C07168=1017.752,24.805,-122.391,-24.214,21.497,-42.553
C07169=1017.754,24.405,-122.357,-24.213,21.497,-42.558
C07170=1017.755,24.022,-122.323,-24.213,21.498,-42.562
C07171=1017.756,23.692,-122.294,-24.213,21.498,-42.564
C07172=1017.757,23.420,-122.270,-24.212,21.498,-42.567
C07173=1017.759,23.186,-122.250,-24.211,21.499,-42.573
C07174=1017.759,22.953,-122.230,-24.211,21.500,-42.577
C07175=1017.760,22.687,-122.207,-24.211,21.500,-42.580
C07176=1017.761,22.366,-122.179,-24.210,21.500,-42.584
C07177=1017.763,21.991,-122.147,-24.210,21.501,-42.586
C07178=1017.764,21.577,-122.111,-24.209,21.501,-42.593
C07179=1017.765,21.333,-122.089,-24.208,21.501,-42.597
C07180=1017.766,21.060,-122.066,-24.208,21.502,-42.599
C07181=1017.767,20.769,-122.041,-24.207,21.501,-42.602
C07182=1017.768,20.472,-122.015,-24.207,21.501,-42.604
C07183=1017.769,20.185,-121.990,-24.207,21.503,-42.606
C07184=1017.770,19.919,-121.966,-24.206,21.502,-42.610
C07185=1017.771,19.682,-121.946,-24.206,21.503,-42.613
C07186=1017.771,19.472,-121.927,-24.205,21.503,-42.617
C07187=1017.773,19.075,-121.894,-24.205,21.503,-42.622
C07188=1017.775,18.678,-121.859,-24.204,21.503,-42.626
C07189=1017.776,18.282,-121.824,-24.203,21.504,-42.632
C07190=1017.777,17.887,-121.790,-24.203,21.505,-42.635
C07191=1017.779,17.493,-121.757,-24.202,21.505,-42.641
C07192=1017.780,17.099,-121.723,-24.201,21.505,-42.646
C07193=1017.781,16.707,-121.689,-24.201,21.506,-42.650
C07194=1017.782,16.316,-121.655,-24.200,21.506,-42.656
C07195=1017.783,15.924,-121.622,-24.200,21.507,-42.659
C07196=1017.785,15.533,-121.587,-24.199,21.507,-42.665
C07197=1017.786,15.145,-121.554,-24.198,21.508,-42.670
C07198=1017.787,14.755,-121.520,-24.198,21.508,-42.674
C07199=1017.788,14.367,-121.487,-24.197,21.509,-42.680
C07200=1017.789,13.980,-121.454,-24.196,21.509,-42.683
C07201=1017.790,13.593,-121.420,-24.196,21.509,-42.689
C07202=1017.792,13.206,-121.387,-24.195,21.511,-42.693
C07203=1017.793,12.819,-121.354,-24.194,21.510,-42.698
C07204=1017.793,12.432,-121.321,-24.193,21.510,-42.703
C07205=1017.795,12.046,-121.287,-24.193,21.512,-42.707
C07206=1017.795,11.659,-121.254,-24.192,21.511,-42.713
C07207=1017.796,11.274,-121.221,-24.192,21.512,-42.716
C07208=1017.798,10.891,-121.188,-24.191,21.513,-42.722
C07209=1017.799,10.510,-121.156,-24.191,21.513,-42.726
C07210=1017.799,10.132,-121.123,-24.190,21.513,-42.731
C07211=1017.800,9.756,-121.091,-24.189,21.514,-42.737
C07212=1017.802,9.379,-121.059,-24.189,21.514,-42.740
C07213=1017.802,9.003,-121.027,-24.188,21.515,-42.746
C07214=1017.804,8.625,-120.994,-24.187,21.515,-42.751
C07215=1017.805,8.245,-120.962,-24.187,21.516,-42.755
C07216=1017.805,7.861,-120.929,-24.186,21.516,-42.761
C07217=1017.806,7.473,-120.896,-24.185,21.517,-42.764
C07218=1017.807,7.082,-120.862,-24.185,21.517,-42.770
C07219=1017.807,6.690,-120.829,-24.184,21.517,-42.775
C07220=1017.809,6.297,-120.796,-24.183,21.519,-42.779
C07221=1017.810,5.903,-120.762,-24.182,21.518,-42.785
C07222=1017.810,5.508,-120.728,-24.182,21.519,-42.790
C07223=1017.811,5.114,-120.695,-24.181,21.520,-42.794
C07224=1017.811,4.719,-120.661,-24.180,21.519,-42.799
C07225=1017.812,4.322,-120.628,-24.180,21.520,-42.805
C07226=1017.814,3.933,-120.595,-24.179,21.521,-42.809
C07227=1017.814,3.574,-120.564,-24.179,21.521,-42.812
C07228=1017.815,3.246,-120.536,-24.178,21.521,-42.817
C07229=1017.815,2.933,-120.509,-24.177,21.522,-42.823
C07230=1017.816,2.610,-120.482,-24.177,21.522,-42.827
C07231=1017.816,2.257,-120.453,-24.176,21.523,-42.833
C07232=1017.817,1.871,-120.419,-24.175,21.524,-42.836
C07233=1017.818,1.474,-120.386,-24.175,21.523,-42.841
C07234=1017.819,1.074,-120.352,-24.174,21.525,-42.846
C07235=1017.818,0.675,-120.318,-24.173,21.525,-42.851
C07236=1017.819,0.273,-120.284,-24.173,21.525,-42.857
C07237=1017.820,-0.130,-120.250,-24.172,21.525,-42.862
C07238=1017.821,-0.537,-120.216,-24.171,21.526,-42.867
C07239=1017.821,-0.945,-120.181,-24.171,21.527,-42.872
C07240=1017.822,-1.354,-120.147,-24.170,21.527,-42.877
C07241=1017.822,-1.767,-120.112,-24.169,21.528,-42.882
C07242=1017.823,-2.182,-120.076,-24.169,21.529,-42.888
C07243=1017.824,-2.599,-120.042,-24.168,21.529,-42.893
C07244=1017.824,-3.018,-120.007,-24.167,21.529,-42.899
C07245=1017.824,-3.439,-119.971,-24.166,21.530,-42.904
C07246=1017.824,-3.651,-119.953,-24.166,21.530,-42.908
C07247=1017.825,-3.863,-119.936,-24.165,21.530,-42.910
C07248=1017.824,-4.077,-119.918,-24.165,21.530,-42.913
C07249=1017.825,-4.292,-119.899,-24.165,21.531,-42.915
C07250=1017.826,-4.508,-119.881,-24.164,21.531,-42.919
C07251=1017.826,-4.727,-119.863,-24.164,21.531,-42.921
C07252=1017.825,-4.947,-119.844,-24.163,21.532,-42.925
C07253=1017.826,-5.169,-119.826,-24.163,21.532,-42.927
C07254=1017.826,-5.391,-119.807,-24.163,21.532,-42.930
C07255=1017.826,-5.615,-119.788,-24.162,21.532,-42.934
C07256=1017.827,-5.838,-119.769,-24.162,21.533,-42.935
C07257=1017.826,-6.064,-119.751,-24.161,21.533,-42.939
C07258=1017.827,-6.287,-119.732,-24.161,21.533,-42.941
C07259=1017.827,-6.511,-119.713,-24.161,21.533,-42.944
C07260=1017.827,-6.735,-119.695,-24.160,21.534,-42.947
C07261=1017.827,-6.957,-119.676,-24.160,21.534,-42.950
C07262=1017.827,-7.178,-119.658,-24.160,21.535,-42.952
C07263=1017.827,-7.399,-119.639,-24.159,21.534,-42.956
C07264=1017.828,-7.618,-119.621,-24.159,21.535,-42.959
C07265=1017.828,-7.836,-119.603,-24.158,21.535,-42.961
C07266=1017.828,-8.053,-119.585,-24.158,21.536,-42.965
C07267=1017.828,-8.270,-119.566,-24.158,21.536,-42.967
C07268=1017.828,-8.487,-119.548,-24.157,21.536,-42.971
C07269=1017.828,-8.703,-119.530,-24.157,21.537,-42.973
C07270=1017.828,-8.919,-119.512,-24.156,21.536,-42.976
C07271=1017.829,-9.136,-119.494,-24.156,21.537,-42.980
C07272=1017.829,-9.353,-119.476,-24.156,21.537,-42.982
C07273=1017.829,-9.569,-119.458,-24.155,21.538,-42.985
C07274=1017.829,-9.786,-119.440,-24.155,21.538,-42.987
C07275=1017.829,-10.001,-119.422,-24.154,21.538,-42.991
C07276=1017.829,-10.217,-119.404,-24.154,21.539,-42.993
C07277=1017.829,-10.432,-119.386,-24.154,21.538,-42.996
C07278=1017.829,-10.647,-119.368,-24.153,21.539,-42.998
C07279=1017.829,-10.861,-119.351,-24.153,21.539,-43.002
C07280=1017.830,-11.076,-119.333,-24.152,21.539,-43.006
C07281=1017.829,-11.290,-119.314,-24.152,21.540,-43.007
C07282=1017.830,-11.503,-119.297,-24.152,21.540,-43.011
C07283=1017.829,-11.715,-119.279,-24.151,21.540,-43.013
C07284=1017.829,-11.928,-119.262,-24.151,21.540,-43.016
C07285=1017.829,-12.140,-119.244,-24.151,21.541,-43.019
C07286=1017.829,-12.351,-119.227,-24.150,21.541,-43.022
C07287=1017.829,-12.562,-119.209,-24.150,21.542,-43.024
C07288=1017.829,-12.982,-119.174,-24.149,21.542,-43.029
C07289=1017.829,-13.400,-119.140,-24.148,21.543,-43.035
C07290=1017.829,-13.813,-119.105,-24.148,21.543,-43.041
C07291=1017.830,-14.226,-119.071,-24.147,21.544,-43.046
C07292=1017.830,-14.634,-119.037,-24.146,21.544,-43.052
C07293=1017.829,-15.039,-119.003,-24.145,21.545,-43.057
C07294=1017.829,-15.442,-118.970,-24.145,21.545,-43.063
C07295=1017.829,-15.843,-118.937,-24.144,21.546,-43.068
C07296=1017.829,-16.242,-118.904,-24.143,21.546,-43.074
C07297=1017.829,-16.642,-118.871,-24.142,21.547,-43.079
C07298=1017.829,-17.039,-118.839,-24.142,21.548,-43.085
C07299=1017.829,-17.437,-118.806,-24.141,21.547,-43.090
C07300=1017.828,-17.847,-118.772,-24.140,21.548,-43.098
C07301=1017.829,-18.096,-118.752,-24.139,21.549,-43.101
C07302=1017.828,-18.384,-118.728,-24.139,21.549,-43.105
C07303=1017.828,-18.695,-118.702,-24.139,21.550,-43.107
C07304=1017.827,-19.006,-118.677,-24.139,21.550,-43.109
C07305=1017.827,-19.294,-118.653,-24.138,21.550,-43.113
C07306=1017.827,-19.543,-118.632,-24.138,21.551,-43.116
C07307=1017.827,-19.954,-118.598,-24.136,21.551,-43.123
C07308=1017.826,-20.352,-118.566,-24.136,21.552,-43.129
C07309=1017.826,-20.749,-118.534,-24.135,21.553,-43.135
C07310=1017.826,-21.147,-118.501,-24.134,21.552,-43.140
C07311=1017.825,-21.545,-118.468,-24.134,21.553,-43.146
C07312=1017.825,-21.942,-118.435,-24.133,21.554,-43.151
C07313=1017.825,-22.340,-118.403,-24.132,21.554,-43.156
C07314=1017.824,-22.737,-118.370,-24.131,21.555,-43.162
C07315=1017.824,-23.135,-118.338,-24.131,21.555,-43.168
C07316=1017.823,-23.532,-118.305,-24.130,21.556,-43.173
C07317=1017.823,-23.929,-118.273,-24.129,21.556,-43.178
C07318=1017.823,-24.327,-118.241,-24.128,21.557,-43.184
C07319=1017.822,-24.725,-118.209,-24.128,21.558,-43.190
C07320=1017.822,-25.122,-118.176,-24.127,21.558,-43.195
C07321=1017.821,-25.520,-118.144,-24.126,21.558,-43.201
C07322=1017.821,-25.918,-118.111,-24.125,21.559,-43.206
C07323=1017.820,-26.315,-118.079,-24.125,21.560,-43.212
C07324=1017.819,-26.712,-118.047,-24.124,21.560,-43.217
C07325=1017.818,-27.109,-118.014,-24.123,21.561,-43.221
C07326=1017.818,-27.507,-117.982,-24.123,21.562,-43.227
C07327=1017.818,-27.904,-117.949,-24.122,21.562,-43.232
C07328=1017.817,-28.301,-117.917,-24.121,21.562,-43.238
C07329=1017.816,-28.700,-117.885,-24.120,21.563,-43.243
C07330=1017.815,-29.097,-117.853,-24.120,21.564,-43.249
C07331=1017.814,-29.494,-117.821,-24.119,21.565,-43.255
C07332=1017.813,-29.892,-117.789,-24.118,21.565,-43.260
C07333=1017.813,-30.289,-117.757,-24.117,21.565,-43.265
C07334=1017.812,-30.686,-117.724,-24.117,21.566,-43.271
C07335=1017.811,-31.083,-117.692,-24.116,21.567,-43.277
C07336=1017.811,-31.481,-117.661,-24.115,21.568,-43.282
C07337=1017.809,-31.879,-117.628,-24.114,21.567,-43.287
C07338=1017.809,-32.276,-117.596,-24.114,21.568,-43.293
C07339=1017.808,-32.674,-117.564,-24.113,21.569,-43.299
C07340=1017.807,-33.071,-117.532,-24.112,21.570,-43.304
C07341=1017.806,-33.469,-117.500,-24.111,21.570,-43.310
C07342=1017.806,-33.866,-117.468,-24.111,21.570,-43.315
C07343=1017.804,-34.263,-117.436,-24.110,21.571,-43.321
C07344=1017.803,-34.660,-117.404,-24.109,21.571,-43.328
C07345=1017.802,-35.058,-117.372,-24.108,21.572,-43.334
C07346=1017.801,-35.456,-117.341,-24.107,21.572,-43.339
C07347=1017.800,-35.853,-117.309,-24.107,21.573,-43.344
C07348=1017.799,-36.250,-117.277,-24.106,21.573,-43.350
C07349=1017.798,-36.647,-117.245,-24.105,21.574,-43.356
C07350=1017.797,-37.044,-117.213,-24.105,21.575,-43.361
C07351=1017.796,-37.442,-117.182,-24.104,21.575,-43.366
C07352=1017.795,-37.839,-117.150,-24.103,21.576,-43.372
C07353=1017.793,-38.237,-117.118,-24.102,21.576,-43.378
C07354=1017.792,-38.634,-117.086,-24.102,21.577,-43.383
C07355=1017.791,-39.032,-117.055,-24.101,21.578,-43.389
C07356=1017.790,-39.429,-117.022,-24.100,21.578,-43.394
C07357=1017.789,-39.826,-116.991,-24.099,21.579,-43.400
C07358=1017.787,-40.223,-116.959,-24.099,21.579,-43.405
C07359=1017.787,-40.621,-116.928,-24.098,21.580,-43.411
C07360=1017.785,-41.017,-116.896,-24.097,21.581,-43.417
C07361=1017.783,-41.415,-116.864,-24.096,21.582,-43.422
C07362=1017.783,-41.813,-116.833,-24.096,21.582,-43.427
C07363=1017.781,-42.210,-116.801,-24.095,21.582,-43.433
C07364=1017.780,-42.607,-116.770,-24.094,21.583,-43.439
C07365=1017.778,-43.004,-116.738,-24.093,21.584,-43.444
C07366=1017.777,-43.401,-116.707,-24.092,21.584,-43.451
C07367=1017.775,-43.798,-116.676,-24.092,21.585,-43.457
C07368=1017.774,-44.195,-116.644,-24.091,21.585,-43.462
C07369=1017.772,-44.593,-116.613,-24.090,21.585,-43.468
C07370=1017.771,-44.990,-116.581,-24.089,21.586,-43.473
C07371=1017.769,-45.387,-116.550,-24.089,21.587,-43.479
C07372=1017.768,-45.785,-116.519,-24.088,21.588,-43.485
C07373=1017.766,-46.182,-116.487,-24.087,21.589,-43.490
C07374=1017.765,-46.579,-116.456,-24.086,21.588,-43.496
C07375=1017.764,-46.976,-116.425,-24.086,21.589,-43.501
C07376=1017.762,-47.373,-116.393,-24.085,21.590,-43.507
C07377=1017.760,-47.770,-116.362,-24.084,21.591,-43.512
C07378=1017.758,-48.167,-116.330,-24.084,21.592,-43.518
C07379=1017.757,-48.565,-116.299,-24.083,21.592,-43.525
C07380=1017.755,-48.962,-116.268,-24.082,21.592,-43.531
C07381=1017.753,-49.358,-116.237,-24.081,21.592,-43.536
C07382=1017.752,-49.756,-116.206,-24.080,21.593,-43.542
C07383=1017.749,-50.153,-116.175,-24.080,21.594,-43.547
C07384=1017.748,-50.550,-116.143,-24.079,21.595,-43.553
C07385=1017.747,-50.947,-116.112,-24.078,21.595,-43.558
C07386=1017.744,-51.344,-116.081,-24.077,21.596,-43.564
C07387=1017.742,-51.740,-116.050,-24.077,21.597,-43.570
C07388=1017.741,-52.138,-116.019,-24.076,21.598,-43.575
C07389=1017.739,-52.534,-115.988,-24.075,21.598,-43.581
C07390=1017.737,-52.931,-115.957,-24.074,21.598,-43.588
C07391=1017.735,-53.328,-115.926,-24.073,21.599,-43.593
C07392=1017.733,-53.725,-115.896,-24.073,21.599,-43.599
C07393=1017.731,-54.122,-115.865,-24.072,21.600,-43.604
C07394=1017.729,-54.519,-115.833,-24.071,21.601,-43.610
C07395=1017.727,-54.916,-115.803,-24.071,21.602,-43.616
C07396=1017.725,-55.313,-115.772,-24.070,21.603,-43.621
C07397=1017.723,-55.711,-115.741,-24.069,21.602,-43.627
C07398=1017.721,-56.108,-115.710,-24.068,21.603,-43.632
C07399=1017.718,-56.505,-115.679,-24.067,21.603,-43.639
C07400=1017.717,-56.904,-115.648,-24.067,21.604,-43.645
C07401=1017.714,-57.302,-115.617,-24.066,21.605,-43.651
C07402=1017.713,-57.701,-115.586,-24.065,21.606,-43.656
C07403=1017.711,-58.100,-115.556,-24.064,21.606,-43.662
C07404=1017.708,-58.500,-115.525,-24.064,21.607,-43.667
C07405=1017.706,-58.900,-115.493,-24.063,21.608,-43.673
C07406=1017.703,-59.300,-115.462,-24.062,21.608,-43.680
C07407=1017.701,-59.702,-115.431,-24.061,21.609,-43.686
C07408=1017.699,-60.104,-115.401,-24.061,21.610,-43.691
C07409=1017.697,-60.506,-115.369,-24.060,21.610,-43.697
C07410=1017.694,-60.909,-115.338,-24.059,21.610,-43.702
C07411=1017.691,-61.313,-115.307,-24.058,21.611,-43.708
C07412=1017.690,-61.717,-115.276,-24.057,21.611,-43.715
C07413=1017.687,-62.121,-115.245,-24.057,21.612,-43.720
C07414=1017.684,-62.527,-115.213,-24.056,21.613,-43.726
C07415=1017.682,-62.932,-115.182,-24.055,21.614,-43.732
C07416=1017.679,-63.339,-115.151,-24.054,21.615,-43.737
C07417=1017.677,-63.745,-115.120,-24.053,21.615,-43.744
C07418=1017.674,-64.153,-115.089,-24.053,21.615,-43.750
C07419=1017.671,-64.560,-115.057,-24.052,21.616,-43.756
C07420=1017.669,-64.969,-115.026,-24.051,21.617,-43.761
C07421=1017.667,-65.377,-114.994,-24.050,21.617,-43.768
C07422=1017.664,-65.786,-114.964,-24.049,21.618,-43.774
C07423=1017.661,-66.195,-114.932,-24.049,21.619,-43.780
C07424=1017.659,-66.604,-114.901,-24.048,21.620,-43.785
C07425=1017.656,-67.014,-114.870,-24.047,21.620,-43.791
C07426=1017.653,-67.424,-114.838,-24.046,21.621,-43.798
C07427=1017.650,-67.834,-114.807,-24.046,21.621,-43.804
C07428=1017.647,-68.244,-114.776,-24.045,21.622,-43.809
C07429=1017.644,-68.655,-114.744,-24.044,21.623,-43.815
C07430=1017.641,-69.066,-114.714,-24.043,21.623,-43.822
C07431=1017.638,-69.476,-114.682,-24.042,21.624,-43.827
C07432=1017.636,-69.888,-114.650,-24.042,21.625,-43.833
C07433=1017.633,-70.298,-114.619,-24.041,21.625,-43.839
C07434=1017.630,-70.710,-114.588,-24.040,21.626,-43.846
C07435=1017.626,-71.121,-114.557,-24.039,21.626,-43.851
C07436=1017.623,-71.532,-114.525,-24.039,21.627,-43.857
C07437=1017.621,-71.942,-114.495,-24.038,21.628,-43.865
C07438=1017.617,-72.353,-114.463,-24.037,21.629,-43.870
C07439=1017.614,-72.764,-114.432,-24.036,21.630,-43.876
C07440=1017.612,-73.175,-114.401,-24.035,21.631,-43.881
C07441=1017.608,-73.586,-114.370,-24.034,21.631,-43.888
C07442=1017.605,-73.996,-114.340,-24.034,21.632,-43.894
C07443=1017.601,-74.407,-114.308,-24.033,21.632,-43.900
C07444=1017.599,-74.817,-114.277,-24.032,21.633,-43.905
C07445=1017.595,-75.226,-114.246,-24.031,21.633,-43.912
C07446=1017.591,-75.636,-114.215,-24.031,21.634,-43.918
C07447=1017.589,-76.046,-114.184,-24.030,21.635,-43.924
C07448=1017.585,-76.456,-114.153,-24.029,21.636,-43.929
C07449=1017.582,-76.865,-114.123,-24.028,21.636,-43.936
C07450=1017.579,-77.273,-114.092,-24.027,21.637,-43.942
C07451=1017.575,-77.681,-114.061,-24.027,21.637,-43.948
C07452=1017.572,-78.090,-114.030,-24.026,21.638,-43.953
C07453=1017.568,-78.497,-114.000,-24.025,21.638,-43.960
C07454=1017.564,-78.905,-113.970,-24.024,21.639,-43.966
C07455=1017.561,-79.311,-113.939,-24.023,21.640,-43.972
C07456=1017.557,-79.718,-113.908,-24.023,21.641,-43.977
C07457=1017.554,-80.124,-113.878,-24.022,21.641,-43.984
C07458=1017.551,-80.528,-113.848,-24.021,21.642,-43.990
C07459=1017.547,-80.932,-113.818,-24.020,21.643,-43.995
C07460=1017.543,-81.337,-113.787,-24.020,21.643,-44.001
C07461=1017.539,-81.739,-113.757,-24.019,21.644,-44.007
C07462=1017.536,-82.142,-113.727,-24.018,21.644,-44.014
C07463=1017.532,-82.545,-113.697,-24.017,21.645,-44.019
C07464=1017.528,-82.946,-113.667,-24.016,21.646,-44.025
C07465=1017.525,-83.347,-113.638,-24.016,21.647,-44.031
C07466=1017.521,-83.747,-113.607,-24.015,21.648,-44.036
C07467=1017.518,-84.148,-113.578,-24.014,21.648,-44.043
C07468=1017.514,-84.553,-113.548,-24.013,21.649,-44.049
C07469=1017.511,-84.777,-113.531,-24.013,21.649,-44.053
C07470=1017.509,-85.018,-113.513,-24.012,21.650,-44.056
C07471=1017.507,-85.271,-113.494,-24.012,21.649,-44.060
C07472=1017.504,-85.526,-113.475,-24.012,21.650,-44.062
C07473=1017.502,-85.772,-113.457,-24.011,21.650,-44.065
C07474=1017.499,-86.001,-113.440,-24.011,21.651,-44.069
C07475=1017.496,-86.411,-113.409,-24.010,21.652,-44.077
C07476=1017.492,-86.799,-113.381,-24.009,21.652,-44.082
C07477=1017.488,-87.179,-113.353,-24.008,21.652,-44.087
C07478=1017.485,-87.551,-113.325,-24.007,21.653,-44.093
C07479=1017.481,-87.923,-113.297,-24.007,21.654,-44.099
C07480=1017.477,-88.299,-113.270,-24.006,21.655,-44.104
C07481=1017.474,-88.706,-113.240,-24.005,21.656,-44.112
C07482=1017.470,-88.954,-113.221,-24.005,21.656,-44.116
C07483=1017.468,-89.228,-113.201,-24.004,21.657,-44.117
C07484=1017.464,-89.512,-113.180,-24.004,21.656,-44.121
C07485=1017.461,-89.787,-113.159,-24.003,21.657,-44.124
C07486=1017.459,-90.037,-113.141,-24.003,21.657,-44.128
C07487=1017.457,-90.256,-113.125,-24.002,21.658,-44.132
C07488=1017.453,-90.652,-113.096,-24.002,21.659,-44.138
C07489=1017.449,-91.045,-113.067,-24.001,21.659,-44.145
C07490=1017.444,-91.438,-113.038,-24.000,21.660,-44.150
C07491=1017.440,-91.830,-113.009,-23.999,21.660,-44.156
C07492=1017.436,-92.222,-112.980,-23.999,21.661,-44.162
C07493=1017.432,-92.612,-112.951,-23.998,21.662,-44.167
C07494=1017.428,-93.002,-112.923,-23.997,21.663,-44.173
C07495=1017.424,-93.391,-112.894,-23.996,21.664,-44.178
C07496=1017.419,-93.780,-112.866,-23.996,21.664,-44.184
C07497=1017.415,-94.168,-112.837,-23.995,21.664,-44.189
C07498=1017.411,-94.554,-112.809,-23.994,21.665,-44.195
C07499=1017.407,-94.941,-112.781,-23.994,21.666,-44.200
C07500=1017.402,-95.326,-112.752,-23.993,21.666,-44.207
C07501=1017.398,-95.711,-112.724,-23.992,21.667,-44.213
C07502=1017.393,-96.096,-112.696,-23.991,21.668,-44.219
C07503=1017.389,-96.480,-112.668,-23.990,21.668,-44.224
C07504=1017.385,-96.863,-112.640,-23.990,21.669,-44.230
C07505=1017.380,-97.247,-112.612,-23.989,21.669,-44.235
C07506=1017.376,-97.630,-112.583,-23.988,21.670,-44.241
C07507=1017.371,-98.014,-112.555,-23.988,21.671,-44.246
C07508=1017.367,-98.396,-112.528,-23.987,21.672,-44.252
C07509=1017.363,-98.780,-112.500,-23.986,21.673,-44.258
C07510=1017.358,-99.164,-112.472,-23.985,21.673,-44.263
C07511=1017.353,-99.547,-112.444,-23.985,21.673,-44.268
C07512=1017.348,-99.932,-112.416,-23.984,21.674,-44.274
C07513=1017.345,-100.316,-112.388,-23.983,21.675,-44.280
C07514=1017.339,-100.701,-112.360,-23.982,21.676,-44.285
C07515=1017.334,-101.086,-112.332,-23.982,21.677,-44.291
C07516=1017.330,-101.473,-112.304,-23.981,21.676,-44.296
C07517=1017.325,-101.861,-112.276,-23.980,21.677,-44.302
C07518=1017.320,-102.248,-112.248,-23.980,21.678,-44.307
C07519=1017.315,-102.636,-112.219,-23.979,21.678,-44.314
C07520=1017.310,-103.026,-112.192,-23.978,21.679,-44.320
C07521=1017.306,-103.416,-112.163,-23.977,21.680,-44.326
C07522=1017.301,-103.806,-112.135,-23.976,21.681,-44.331
C07523=1017.296,-104.197,-112.106,-23.976,21.682,-44.337
C07524=1017.290,-104.588,-112.078,-23.975,21.681,-44.342
C07525=1017.285,-104.981,-112.050,-23.974,21.682,-44.348
C07526=1017.280,-105.373,-112.022,-23.974,21.683,-44.353
C07527=1017.275,-105.765,-111.993,-23.973,21.684,-44.359
C07528=1017.270,-106.158,-111.965,-23.972,21.685,-44.365
C07529=1017.265,-106.552,-111.936,-23.971,21.686,-44.370
C07530=1017.260,-106.944,-111.907,-23.971,21.686,-44.376
C07531=1017.255,-107.337,-111.879,-23.970,21.687,-44.383
C07532=1017.249,-107.730,-111.851,-23.969,21.687,-44.388
C07533=1017.244,-108.123,-111.822,-23.968,21.688,-44.394
C07534=1017.238,-108.516,-111.794,-23.968,21.688,-44.399
C07535=1017.233,-108.909,-111.766,-23.967,21.689,-44.405
C07536=1017.227,-109.301,-111.738,-23.966,21.690,-44.411
C07537=1017.222,-109.695,-111.710,-23.965,21.691,-44.416
C07538=1017.217,-110.088,-111.682,-23.965,21.691,-44.422
C07539=1017.211,-110.481,-111.653,-23.964,21.692,-44.427
C07540=1017.205,-110.873,-111.625,-23.963,21.693,-44.433
C07541=1017.199,-111.266,-111.596,-23.963,21.694,-44.439
C07542=1017.194,-111.659,-111.568,-23.962,21.694,-44.446
C07543=1017.188,-112.051,-111.540,-23.961,21.694,-44.451
C07544=1017.183,-112.444,-111.512,-23.960,21.695,-44.456
C07545=1017.177,-112.836,-111.484,-23.959,21.696,-44.462
C07546=1017.172,-113.229,-111.456,-23.959,21.696,-44.468
C07547=1017.165,-113.622,-111.428,-23.958,21.697,-44.473
C07548=1017.160,-114.015,-111.400,-23.957,21.698,-44.479
C07549=1017.154,-114.407,-111.371,-23.957,21.699,-44.485
C07550=1017.148,-114.800,-111.344,-23.956,21.700,-44.490
C07551=1017.143,-115.192,-111.315,-23.955,21.701,-44.496
C07552=1017.137,-115.584,-111.287,-23.954,21.700,-44.501
C07553=1017.131,-115.977,-111.260,-23.954,21.701,-44.507
C07554=1017.125,-116.369,-111.232,-23.953,21.702,-44.512
C07555=1017.118,-116.762,-111.203,-23.952,21.703,-44.518
C07556=1017.113,-117.154,-111.176,-23.952,21.704,-44.523
C07557=1017.107,-117.546,-111.148,-23.951,21.705,-44.529
C07558=1017.100,-117.938,-111.120,-23.950,21.705,-44.536
C07559=1017.095,-118.331,-111.092,-23.949,21.705,-44.541
C07560=1017.089,-118.723,-111.064,-23.948,21.706,-44.547
C07561=1017.082,-119.115,-111.036,-23.948,21.706,-44.553
C07562=1017.077,-119.508,-111.009,-23.947,21.707,-44.558
C07563=1017.070,-119.900,-110.980,-23.946,21.708,-44.564
C07564=1017.064,-120.292,-110.952,-23.946,21.709,-44.569
C07565=1017.057,-120.684,-110.924,-23.945,21.710,-44.575
C07566=1017.051,-121.077,-110.897,-23.944,21.710,-44.580
C07567=1017.045,-121.469,-110.869,-23.943,21.710,-44.586
C07568=1017.039,-121.861,-110.841,-23.943,21.711,-44.591
C07569=1017.032,-122.253,-110.813,-23.942,21.712,-44.597
C07570=1017.026,-122.645,-110.785,-23.941,21.713,-44.603
C07571=1017.019,-123.037,-110.757,-23.941,21.714,-44.608
C07572=1017.013,-123.430,-110.730,-23.940,21.715,-44.614
C07573=1017.006,-123.821,-110.702,-23.939,21.714,-44.619
C07574=1017.000,-124.214,-110.674,-23.939,21.715,-44.625
C07575=1016.993,-124.605,-110.647,-23.938,21.716,-44.630
C07576=1016.986,-124.997,-110.619,-23.937,21.717,-44.636
C07577=1016.979,-125.390,-110.591,-23.936,21.718,-44.642
C07578=1016.973,-125.753,-110.566,-23.936,21.718,-44.647
C07579=1016.966,-126.173,-110.536,-23.935,21.719,-44.652
C07580=1016.959,-126.565,-110.508,-23.934,21.719,-44.658
C07581=1016.953,-126.957,-110.480,-23.934,21.720,-44.664
C07582=1016.946,-127.349,-110.452,-23.933,21.721,-44.669
C07583=1016.939,-127.742,-110.425,-23.932,21.722,-44.675
C07584=1016.932,-128.133,-110.398,-23.932,21.723,-44.680
C07585=1016.925,-128.525,-110.370,-23.931,21.723,-44.686
C07586=1016.918,-128.917,-110.343,-23.930,21.723,-44.691
C07587=1016.911,-129.309,-110.315,-23.929,21.724,-44.697
C07588=1016.904,-129.701,-110.287,-23.929,21.725,-44.703
C07589=1016.897,-130.093,-110.260,-23.928,21.726,-44.708
C07590=1016.890,-130.484,-110.232,-23.927,21.727,-44.714
C07591=1016.882,-130.876,-110.204,-23.926,21.727,-44.719
C07592=1016.875,-131.268,-110.177,-23.926,21.728,-44.725
C07593=1016.868,-131.659,-110.149,-23.925,21.728,-44.730
C07594=1016.861,-132.052,-110.121,-23.924,21.729,-44.736
C07595=1016.853,-132.443,-110.094,-23.924,21.730,-44.741
C07596=1016.846,-132.835,-110.067,-23.923,21.730,-44.747
C07597=1016.839,-133.227,-110.039,-23.922,21.731,-44.752
C07598=1016.831,-133.619,-110.012,-23.922,21.732,-44.758
C07599=1016.825,-134.011,-109.984,-23.921,21.732,-44.763
C07600=1017.216,-133.982,-110.228,-23.921,21.732,-44.763
C07601=1017.222,-133.590,-110.256,-23.922,21.732,-44.758
C07602=1017.230,-133.199,-110.283,-23.922,21.731,-44.752
C07603=1017.237,-132.807,-110.310,-23.923,21.730,-44.747
C07604=1017.244,-132.415,-110.338,-23.924,21.730,-44.741
C07605=1017.252,-132.023,-110.365,-23.924,21.729,-44.736
C07606=1017.259,-131.632,-110.393,-23.925,21.728,-44.730
C07607=1017.266,-131.240,-110.420,-23.926,21.728,-44.725
C07608=1017.272,-130.848,-110.448,-23.926,21.727,-44.719
C07609=1017.279,-130.456,-110.475,-23.927,21.727,-44.714
C07610=1017.286,-130.064,-110.502,-23.928,21.726,-44.708
C07611=1017.293,-129.672,-110.530,-23.929,21.725,-44.703
C07612=1017.299,-129.281,-110.557,-23.929,21.724,-44.697
C07613=1017.306,-128.889,-110.585,-23.930,21.723,-44.691
C07614=1017.314,-128.497,-110.613,-23.931,21.723,-44.686
C07615=1017.321,-128.105,-110.640,-23.932,21.723,-44.680
C07616=1017.327,-127.713,-110.667,-23.932,21.722,-44.675
C07617=1017.334,-127.321,-110.694,-23.933,21.721,-44.669
C07618=1017.341,-126.929,-110.722,-23.934,21.720,-44.664
C07619=1017.347,-126.537,-110.750,-23.934,21.719,-44.658
C07620=1017.354,-126.145,-110.778,-23.935,21.719,-44.652
C07621=1017.360,-125.753,-110.804,-23.936,21.719,-44.647
C07622=1017.366,-125.361,-110.832,-23.936,21.718,-44.642
C07623=1017.373,-124.969,-110.860,-23.937,21.717,-44.636
C07624=1017.380,-124.577,-110.888,-23.938,21.716,-44.630
C07625=1017.386,-124.185,-110.916,-23.939,21.715,-44.625
C07626=1017.393,-123.793,-110.942,-23.939,21.714,-44.619
C07627=1017.399,-123.401,-110.971,-23.940,21.715,-44.614
C07628=1017.406,-123.009,-110.998,-23.941,21.714,-44.608
C07629=1017.411,-122.617,-111.026,-23.941,21.713,-44.603
C07630=1017.418,-122.225,-111.054,-23.942,21.712,-44.597
C07631=1017.424,-121.833,-111.081,-23.943,21.711,-44.591
C07632=1017.430,-121.441,-111.109,-23.943,21.710,-44.586
C07633=1017.436,-121.048,-111.137,-23.944,21.710,-44.580
C07634=1017.442,-120.656,-111.165,-23.945,21.710,-44.575
C07635=1017.449,-120.264,-111.192,-23.946,21.709,-44.569
C07636=1017.455,-119.872,-111.220,-23.946,21.708,-44.564
C07637=1017.461,-119.480,-111.248,-23.947,21.707,-44.558
C07638=1017.467,-119.087,-111.275,-23.948,21.706,-44.553
C07639=1017.473,-118.695,-111.303,-23.948,21.706,-44.547
C07640=1017.479,-118.303,-111.332,-23.949,21.705,-44.541
C07641=1017.484,-117.911,-111.359,-23.950,21.705,-44.536
C07642=1017.490,-117.519,-111.387,-23.951,21.705,-44.529
C07643=1017.496,-117.126,-111.414,-23.952,21.704,-44.523
C07644=1017.502,-116.734,-111.442,-23.952,21.703,-44.518
C07645=1017.508,-116.342,-111.470,-23.953,21.702,-44.512
C07646=1017.513,-115.949,-111.498,-23.954,21.701,-44.507
C07647=1017.519,-115.557,-111.526,-23.954,21.700,-44.501
C07648=1017.525,-115.165,-111.554,-23.955,21.701,-44.496
C07649=1017.530,-114.772,-111.582,-23.956,21.700,-44.490
C07650=1017.536,-114.380,-111.610,-23.957,21.699,-44.485
C07651=1017.542,-113.987,-111.637,-23.957,21.698,-44.479
C07652=1017.548,-113.595,-111.666,-23.958,21.697,-44.473
C07653=1017.553,-113.202,-111.694,-23.959,21.696,-44.468
C07654=1017.559,-112.810,-111.722,-23.959,21.696,-44.462
C07655=1017.565,-112.416,-111.750,-23.960,21.695,-44.456
C07656=1017.571,-112.024,-111.779,-23.961,21.694,-44.451
C07657=1017.576,-111.631,-111.807,-23.962,21.694,-44.446
C07658=1017.581,-111.238,-111.834,-23.963,21.694,-44.439
C07659=1017.587,-110.846,-111.863,-23.963,21.693,-44.433
C07660=1017.592,-110.453,-111.891,-23.964,21.692,-44.427
C07661=1017.598,-110.060,-111.918,-23.965,21.691,-44.422
C07662=1017.603,-109.668,-111.947,-23.965,21.691,-44.416
C07663=1017.608,-109.275,-111.975,-23.966,21.690,-44.411
C07664=1017.613,-108.882,-112.003,-23.967,21.689,-44.405
C07665=1017.618,-108.489,-112.031,-23.968,21.688,-44.399
C07666=1017.624,-108.096,-112.060,-23.968,21.688,-44.394
C07667=1017.629,-107.703,-112.088,-23.969,21.687,-44.388
C07668=1017.634,-107.310,-112.116,-23.970,21.687,-44.383
C07669=1017.639,-106.917,-112.144,-23.971,21.686,-44.376
C07670=1017.644,-106.524,-112.172,-23.971,21.686,-44.370
C07671=1017.650,-106.132,-112.201,-23.972,21.685,-44.365
C07672=1017.654,-105.738,-112.229,-23.973,21.684,-44.359
C07673=1017.659,-105.345,-112.257,-23.974,21.683,-44.353
C07674=1017.664,-104.953,-112.286,-23.974,21.682,-44.348
C07675=1017.669,-104.561,-112.314,-23.975,21.681,-44.342
C07676=1017.675,-104.170,-112.342,-23.976,21.682,-44.337
C07677=1017.679,-103.778,-112.371,-23.976,21.681,-44.331
C07678=1017.684,-103.388,-112.399,-23.977,21.680,-44.326
C07679=1017.689,-102.999,-112.427,-23.978,21.679,-44.320
C07680=1017.694,-102.609,-112.455,-23.979,21.678,-44.314
C07681=1017.698,-102.221,-112.483,-23.980,21.678,-44.307
C07682=1017.702,-101.833,-112.511,-23.980,21.677,-44.302
C07683=1017.708,-101.446,-112.539,-23.981,21.676,-44.296
C07684=1017.713,-101.060,-112.567,-23.982,21.677,-44.291
C07685=1017.717,-100.673,-112.595,-23.982,21.676,-44.285
C07686=1017.722,-100.288,-112.623,-23.983,21.675,-44.280
C07687=1017.726,-99.904,-112.651,-23.984,21.674,-44.274
C07688=1017.731,-99.520,-112.679,-23.985,21.673,-44.268
C07689=1017.735,-99.136,-112.707,-23.985,21.673,-44.263
C07690=1017.740,-98.753,-112.735,-23.986,21.673,-44.258
C07691=1017.744,-98.370,-112.763,-23.987,21.672,-44.252
C07692=1017.748,-97.986,-112.791,-23.988,21.671,-44.246
C07693=1017.753,-97.603,-112.819,-23.988,21.670,-44.241
C07694=1017.757,-97.220,-112.847,-23.989,21.669,-44.235
C07695=1017.762,-96.836,-112.875,-23.990,21.669,-44.230
C07696=1017.765,-96.452,-112.903,-23.990,21.668,-44.224
C07697=1017.770,-96.069,-112.930,-23.991,21.668,-44.219
C07698=1017.775,-95.684,-112.959,-23.992,21.667,-44.213
C07699=1017.779,-95.299,-112.987,-23.993,21.666,-44.207
C07700=1017.783,-94.913,-113.015,-23.994,21.666,-44.200
C07701=1017.787,-94.527,-113.043,-23.994,21.665,-44.195
C07702=1017.791,-94.140,-113.072,-23.995,21.664,-44.189
C07703=1017.795,-93.753,-113.101,-23.996,21.664,-44.184
C07704=1017.800,-93.365,-113.129,-23.996,21.664,-44.178
C07705=1017.804,-92.975,-113.157,-23.997,21.663,-44.173
C07706=1017.808,-92.585,-113.186,-23.998,21.662,-44.167
C07707=1017.813,-92.194,-113.214,-23.999,21.661,-44.162
C07708=1017.816,-91.803,-113.243,-23.999,21.660,-44.156
C07709=1017.820,-91.411,-113.272,-24.000,21.660,-44.150
C07710=1017.824,-91.018,-113.301,-24.001,21.659,-44.145
C07711=1017.828,-90.624,-113.330,-24.002,21.659,-44.138
C07712=1017.832,-90.229,-113.359,-24.002,21.658,-44.132
C07713=1017.835,-90.010,-113.375,-24.003,21.657,-44.128
C07714=1017.837,-89.760,-113.393,-24.003,21.657,-44.124
C07715=1017.840,-89.485,-113.414,-24.004,21.656,-44.121
C07716=1017.843,-89.200,-113.435,-24.004,21.657,-44.117
C07717=1017.845,-88.926,-113.455,-24.005,21.656,-44.116
C07718=1017.848,-88.679,-113.473,-24.005,21.656,-44.112
C07719=1017.852,-88.271,-113.503,-24.006,21.655,-44.104
C07720=1017.855,-87.896,-113.531,-24.007,21.654,-44.099
C07721=1017.859,-87.524,-113.559,-24.007,21.653,-44.093
C07722=1017.863,-87.151,-113.586,-24.008,21.652,-44.087
C07723=1017.866,-86.772,-113.614,-24.009,21.652,-44.082
C07724=1017.870,-86.384,-113.643,-24.010,21.652,-44.077
C07725=1017.874,-85.975,-113.673,-24.011,21.651,-44.069
C07726=1017.876,-85.745,-113.690,-24.011,21.650,-44.065
C07727=1017.878,-85.499,-113.708,-24.012,21.650,-44.062
C07728=1017.881,-85.244,-113.727,-24.012,21.649,-44.060
C07729=1017.883,-84.991,-113.746,-24.012,21.650,-44.056
C07730=1017.885,-84.750,-113.764,-24.013,21.649,-44.053
C07731=1017.887,-84.527,-113.781,-24.013,21.649,-44.049
C07732=1017.891,-84.120,-113.811,-24.014,21.648,-44.043
C07733=1017.895,-83.721,-113.840,-24.015,21.648,-44.036
C07734=1017.898,-83.320,-113.870,-24.016,21.647,-44.031
C07735=1017.902,-82.919,-113.900,-24.016,21.646,-44.025
C07736=1017.906,-82.518,-113.930,-24.017,21.645,-44.019
C07737=1017.910,-82.116,-113.960,-24.018,21.644,-44.014
C07738=1017.913,-81.713,-113.990,-24.019,21.644,-44.007
C07739=1017.917,-81.310,-114.020,-24.020,21.643,-44.001
C07740=1017.920,-80.905,-114.050,-24.020,21.643,-43.995
C07741=1017.924,-80.501,-114.080,-24.021,21.642,-43.990
C07742=1017.927,-80.096,-114.111,-24.022,21.641,-43.984
C07743=1017.930,-79.691,-114.141,-24.023,21.641,-43.977
C07744=1017.934,-79.284,-114.172,-24.023,21.640,-43.972
C07745=1017.937,-78.878,-114.202,-24.024,21.639,-43.966
C07746=1017.941,-78.470,-114.232,-24.025,21.638,-43.960
C07747=1017.945,-78.062,-114.263,-24.026,21.638,-43.953
C07748=1017.947,-77.655,-114.293,-24.027,21.637,-43.948
C07749=1017.951,-77.246,-114.324,-24.027,21.637,-43.942
C07750=1017.954,-76.837,-114.355,-24.028,21.636,-43.936
C07751=1017.957,-76.428,-114.386,-24.029,21.636,-43.929
C07752=1017.960,-76.019,-114.417,-24.030,21.635,-43.924
C07753=1017.964,-75.610,-114.447,-24.031,21.634,-43.918
C07754=1017.968,-75.200,-114.478,-24.031,21.633,-43.912
C07755=1017.970,-74.790,-114.509,-24.032,21.633,-43.905
C07756=1017.973,-74.379,-114.540,-24.033,21.632,-43.900
C07757=1017.977,-73.969,-114.571,-24.034,21.632,-43.894
C07758=1017.980,-73.559,-114.602,-24.034,21.631,-43.888
C07759=1017.983,-73.148,-114.633,-24.035,21.631,-43.881
C07760=1017.985,-72.737,-114.664,-24.036,21.630,-43.876
C07761=1017.989,-72.326,-114.696,-24.037,21.629,-43.870
C07762=1017.992,-71.915,-114.727,-24.038,21.628,-43.865
C07763=1017.995,-71.504,-114.757,-24.039,21.627,-43.857
C07764=1017.998,-71.094,-114.789,-24.039,21.626,-43.851
C07765=1018.001,-70.682,-114.820,-24.040,21.626,-43.846
C07766=1018.004,-70.272,-114.850,-24.041,21.625,-43.839
C07767=1018.007,-69.861,-114.882,-24.042,21.625,-43.833
C07768=1018.010,-69.450,-114.913,-24.042,21.624,-43.827
C07769=1018.013,-69.039,-114.944,-24.043,21.623,-43.822
C07770=1018.015,-68.628,-114.976,-24.044,21.623,-43.815
C07771=1018.018,-68.218,-115.007,-24.045,21.622,-43.809
C07772=1018.021,-67.808,-115.039,-24.046,21.621,-43.804
C07773=1018.023,-67.397,-115.069,-24.046,21.621,-43.798
C07774=1018.026,-66.987,-115.101,-24.047,21.620,-43.791
C07775=1018.029,-66.578,-115.133,-24.048,21.620,-43.785
C07776=1018.032,-66.168,-115.164,-24.049,21.619,-43.780
C07777=1018.034,-65.758,-115.195,-24.049,21.618,-43.774
C07778=1018.038,-65.350,-115.226,-24.050,21.617,-43.768
C07779=1018.040,-64.942,-115.257,-24.051,21.617,-43.761
C07780=1018.042,-64.533,-115.289,-24.052,21.616,-43.756
C07781=1018.045,-64.126,-115.320,-24.053,21.615,-43.750
C07782=1018.048,-63.719,-115.351,-24.053,21.615,-43.744
C07783=1018.050,-63.313,-115.382,-24.054,21.615,-43.737
C07784=1018.053,-62.906,-115.413,-24.055,21.614,-43.732
C07785=1018.055,-62.500,-115.444,-24.056,21.613,-43.726
C07786=1018.057,-62.095,-115.476,-24.057,21.612,-43.720
C07787=1018.060,-61.690,-115.506,-24.057,21.611,-43.715
C07788=1018.062,-61.285,-115.538,-24.058,21.611,-43.708
C07789=1018.065,-60.882,-115.569,-24.059,21.610,-43.702
C07790=1018.066,-60.479,-115.600,-24.060,21.610,-43.697
C07791=1018.069,-60.077,-115.631,-24.061,21.610,-43.691
C07792=1018.071,-59.675,-115.661,-24.061,21.609,-43.686
C07793=1018.073,-59.274,-115.693,-24.062,21.608,-43.680
C07794=1018.076,-58.874,-115.724,-24.063,21.608,-43.673
C07795=1018.078,-58.473,-115.755,-24.064,21.607,-43.667
C07796=1018.080,-58.074,-115.786,-24.064,21.606,-43.662
C07797=1018.083,-57.674,-115.817,-24.065,21.606,-43.656
C07798=1018.084,-57.275,-115.847,-24.066,21.605,-43.651
C07799=1018.087,-56.877,-115.878,-24.067,21.604,-43.645
C07800=1018.088,-56.479,-115.909,-24.067,21.603,-43.639
C07801=1018.091,-56.081,-115.940,-24.068,21.603,-43.632
C07802=1018.092,-55.683,-115.971,-24.069,21.602,-43.627
C07803=1018.095,-55.286,-116.002,-24.070,21.603,-43.621
C07804=1018.097,-54.889,-116.032,-24.071,21.602,-43.616
C07805=1018.098,-54.492,-116.064,-24.071,21.601,-43.610
C07806=1018.101,-54.095,-116.095,-24.072,21.600,-43.604
C07807=1018.103,-53.698,-116.125,-24.073,21.599,-43.599
C07808=1018.104,-53.301,-116.157,-24.073,21.599,-43.593
C07809=1018.106,-52.905,-116.188,-24.074,21.598,-43.588
C07810=1018.108,-52.507,-116.218,-24.075,21.598,-43.581
C07811=1018.110,-52.110,-116.250,-24.076,21.598,-43.575
C07812=1018.112,-51.714,-116.281,-24.077,21.597,-43.570
C07813=1018.114,-51.317,-116.311,-24.077,21.596,-43.564
C07814=1018.116,-50.920,-116.343,-24.078,21.595,-43.558
C07815=1018.117,-50.523,-116.374,-24.079,21.595,-43.553
C07816=1018.119,-50.126,-116.405,-24.080,21.594,-43.547
C07817=1018.121,-49.729,-116.436,-24.080,21.593,-43.542
C07818=1018.123,-49.332,-116.467,-24.081,21.592,-43.536
C07819=1018.124,-48.934,-116.498,-24.082,21.592,-43.531
C07820=1018.125,-48.537,-116.530,-24.083,21.592,-43.525
C07821=1018.128,-48.141,-116.561,-24.084,21.592,-43.518
C07822=1018.129,-47.743,-116.591,-24.084,21.591,-43.512
C07823=1018.130,-47.346,-116.623,-24.085,21.590,-43.507
C07824=1018.132,-46.949,-116.655,-24.086,21.589,-43.501
C07825=1018.133,-46.552,-116.685,-24.086,21.588,-43.496
C07826=1018.135,-46.155,-116.717,-24.087,21.589,-43.490
C07827=1018.137,-45.758,-116.748,-24.088,21.588,-43.485
C07828=1018.138,-45.361,-116.779,-24.089,21.587,-43.479
C07829=1018.140,-44.964,-116.811,-24.089,21.586,-43.473
C07830=1018.142,-44.566,-116.842,-24.090,21.585,-43.468
C07831=1018.143,-44.169,-116.873,-24.091,21.585,-43.462
C07832=1018.144,-43.772,-116.905,-24.092,21.585,-43.457
C07833=1018.145,-43.375,-116.937,-24.092,21.584,-43.451
C07834=1018.146,-42.977,-116.968,-24.093,21.584,-43.444
C07835=1018.148,-42.580,-117.000,-24.094,21.583,-43.439
C07836=1018.149,-42.183,-117.031,-24.095,21.582,-43.433
C07837=1018.151,-41.786,-117.062,-24.096,21.582,-43.427
C07838=1018.152,-41.389,-117.094,-24.096,21.582,-43.422
C07839=1018.153,-40.991,-117.126,-24.097,21.581,-43.417
C07840=1018.154,-40.595,-117.157,-24.098,21.580,-43.411
C07841=1018.156,-40.196,-117.189,-24.099,21.579,-43.405
C07842=1018.157,-39.799,-117.221,-24.099,21.579,-43.400
C07843=1018.159,-39.402,-117.252,-24.100,21.578,-43.394
C07844=1018.160,-39.005,-117.283,-24.101,21.578,-43.389
C07845=1018.160,-38.607,-117.315,-24.102,21.577,-43.383
C07846=1018.162,-38.210,-117.347,-24.102,21.576,-43.378
C07847=1018.163,-37.813,-117.379,-24.103,21.576,-43.372
C07848=1018.164,-37.416,-117.410,-24.104,21.575,-43.366
C07849=1018.165,-37.018,-117.442,-24.105,21.575,-43.361
C07850=1018.166,-36.620,-117.475,-24.105,21.574,-43.356
C07851=1018.168,-36.223,-117.506,-24.106,21.573,-43.350
C07852=1018.168,-35.826,-117.538,-24.107,21.573,-43.344
C07853=1018.170,-35.429,-117.570,-24.107,21.572,-43.339
C07854=1018.170,-35.031,-117.602,-24.108,21.572,-43.334
C07855=1018.171,-34.634,-117.634,-24.109,21.571,-43.328
C07856=1018.172,-34.236,-117.665,-24.110,21.571,-43.321
C07857=1018.173,-33.839,-117.697,-24.111,21.570,-43.315
C07858=1018.174,-33.442,-117.729,-24.111,21.570,-43.310
C07859=1018.175,-33.044,-117.762,-24.112,21.570,-43.304
C07860=1018.176,-32.647,-117.794,-24.113,21.569,-43.299
C07861=1018.176,-32.249,-117.825,-24.114,21.568,-43.293
C07862=1018.177,-31.852,-117.858,-24.114,21.567,-43.287
C07863=1018.178,-31.455,-117.890,-24.115,21.568,-43.282
C07864=1018.179,-31.057,-117.922,-24.116,21.567,-43.277
C07865=1018.180,-30.660,-117.954,-24.117,21.566,-43.271
C07866=1018.180,-30.263,-117.986,-24.117,21.565,-43.265
C07867=1018.181,-29.865,-118.018,-24.118,21.565,-43.260
C07868=1018.182,-29.467,-118.050,-24.119,21.565,-43.255
C07869=1018.183,-29.070,-118.082,-24.120,21.564,-43.249
C07870=1018.184,-28.673,-118.115,-24.120,21.563,-43.243
C07871=1018.184,-28.275,-118.147,-24.121,21.562,-43.238
C07872=1018.185,-27.878,-118.179,-24.122,21.562,-43.232
C07873=1018.186,-27.481,-118.211,-24.123,21.562,-43.227
C07874=1018.186,-27.083,-118.243,-24.123,21.561,-43.221
C07875=1018.187,-26.685,-118.275,-24.124,21.560,-43.217
C07876=1018.187,-26.288,-118.308,-24.125,21.560,-43.212
C07877=1018.187,-25.891,-118.340,-24.125,21.559,-43.206
C07878=1018.189,-25.493,-118.373,-24.126,21.558,-43.201
C07879=1018.189,-25.095,-118.405,-24.127,21.558,-43.195
C07880=1018.189,-24.698,-118.438,-24.128,21.558,-43.190
C07881=1018.190,-24.301,-118.470,-24.128,21.557,-43.184
C07882=1018.191,-23.903,-118.502,-24.129,21.556,-43.178
C07883=1018.191,-23.506,-118.535,-24.130,21.556,-43.173
C07884=1018.192,-23.109,-118.567,-24.131,21.555,-43.168
C07885=1018.192,-22.711,-118.600,-24.131,21.555,-43.162
C07886=1018.192,-22.313,-118.632,-24.132,21.554,-43.156
C07887=1018.192,-21.916,-118.664,-24.133,21.554,-43.151
C07888=1018.192,-21.518,-118.697,-24.134,21.553,-43.146
C07889=1018.194,-21.120,-118.730,-24.134,21.552,-43.140
C07890=1018.194,-20.723,-118.762,-24.135,21.553,-43.135
C07891=1018.194,-20.325,-118.795,-24.136,21.552,-43.129
C07892=1018.195,-19.928,-118.827,-24.136,21.551,-43.123
C07893=1018.195,-19.517,-118.862,-24.138,21.551,-43.116
C07894=1018.195,-19.268,-118.882,-24.138,21.550,-43.113
C07895=1018.195,-18.979,-118.906,-24.139,21.550,-43.109
C07896=1018.195,-18.668,-118.931,-24.139,21.550,-43.107
C07897=1018.195,-18.357,-118.957,-24.139,21.549,-43.105
C07898=1018.195,-18.070,-118.980,-24.139,21.549,-43.101
C07899=1018.196,-17.821,-119.002,-24.140,21.548,-43.098
C07900=1018.196,-17.410,-119.035,-24.141,21.547,-43.090
C07901=1018.196,-17.012,-119.067,-24.142,21.548,-43.085
C07902=1018.196,-16.615,-119.100,-24.142,21.547,-43.079
C07903=1018.196,-16.216,-119.133,-24.143,21.546,-43.074
C07904=1018.197,-15.816,-119.166,-24.144,21.546,-43.068
C07905=1018.196,-15.415,-119.199,-24.145,21.545,-43.063
C07906=1018.196,-15.012,-119.233,-24.145,21.545,-43.057
C07907=1018.196,-14.607,-119.266,-24.146,21.544,-43.052
C07908=1018.196,-14.199,-119.300,-24.147,21.544,-43.046
C07909=1018.197,-13.787,-119.334,-24.148,21.543,-43.041
C07910=1018.197,-13.373,-119.369,-24.148,21.543,-43.035
C07911=1018.197,-12.955,-119.403,-24.149,21.542,-43.029
C07912=1018.197,-12.535,-119.438,-24.150,21.542,-43.024
C07913=1018.196,-12.324,-119.455,-24.150,21.541,-43.022
C07914=1018.197,-12.113,-119.473,-24.151,21.541,-43.019
C07915=1018.197,-11.902,-119.491,-24.151,21.540,-43.016
C07916=1018.197,-11.689,-119.508,-24.151,21.540,-43.013
C07917=1018.196,-11.476,-119.526,-24.152,21.540,-43.011
C07918=1018.196,-11.263,-119.544,-24.152,21.540,-43.007
C07919=1018.197,-11.049,-119.562,-24.152,21.539,-43.006
C07920=1018.197,-10.835,-119.580,-24.153,21.539,-43.002
C07921=1018.197,-10.620,-119.597,-24.153,21.539,-42.998
C07922=1018.196,-10.406,-119.615,-24.154,21.538,-42.996
C07923=1018.196,-10.190,-119.633,-24.154,21.539,-42.993
C07924=1018.196,-9.975,-119.650,-24.154,21.538,-42.991
C07925=1018.196,-9.759,-119.669,-24.155,21.538,-42.987
C07926=1018.196,-9.543,-119.687,-24.155,21.538,-42.985
C07927=1018.196,-9.327,-119.705,-24.156,21.537,-42.982
C07928=1018.196,-9.109,-119.723,-24.156,21.537,-42.980
C07929=1018.195,-8.893,-119.741,-24.156,21.536,-42.976
C07930=1018.195,-8.677,-119.759,-24.157,21.537,-42.973
C07931=1018.196,-8.460,-119.777,-24.157,21.536,-42.971
C07932=1018.195,-8.243,-119.796,-24.158,21.536,-42.967
C07933=1018.195,-8.026,-119.814,-24.158,21.536,-42.965
C07934=1018.196,-7.810,-119.832,-24.158,21.535,-42.961
C07935=1018.195,-7.591,-119.850,-24.159,21.535,-42.959
C07936=1018.195,-7.372,-119.868,-24.159,21.534,-42.956
C07937=1018.195,-7.151,-119.887,-24.160,21.535,-42.952
C07938=1018.194,-6.930,-119.905,-24.160,21.534,-42.950
C07939=1018.195,-6.708,-119.923,-24.160,21.534,-42.947
C07940=1018.194,-6.484,-119.942,-24.161,21.533,-42.944
C07941=1018.194,-6.261,-119.961,-24.161,21.533,-42.941
C07942=1018.194,-6.037,-119.980,-24.161,21.533,-42.939
C07943=1018.194,-5.812,-119.998,-24.162,21.533,-42.935
C07944=1018.194,-5.588,-120.017,-24.162,21.532,-42.934
C07945=1018.193,-5.364,-120.036,-24.163,21.532,-42.930
C07946=1018.193,-5.142,-120.055,-24.163,21.532,-42.927
C07947=1018.193,-4.921,-120.073,-24.163,21.532,-42.925
C07948=1018.192,-4.701,-120.092,-24.164,21.531,-42.921
C07949=1018.192,-4.482,-120.110,-24.164,21.531,-42.919
C07950=1018.192,-4.265,-120.128,-24.165,21.531,-42.915
C07951=1018.192,-4.050,-120.147,-24.165,21.530,-42.913
C07952=1018.192,-3.837,-120.164,-24.165,21.530,-42.910
C07953=1018.191,-3.624,-120.182,-24.166,21.530,-42.908
C07954=1018.192,-3.413,-120.200,-24.166,21.530,-42.904
C07955=1018.190,-2.992,-120.235,-24.167,21.529,-42.899
C07956=1018.190,-2.572,-120.271,-24.168,21.529,-42.893
C07957=1018.189,-2.155,-120.306,-24.169,21.529,-42.888
C07958=1018.189,-1.740,-120.341,-24.169,21.528,-42.882
C07959=1018.189,-1.328,-120.376,-24.170,21.527,-42.877
C07960=1018.188,-0.918,-120.411,-24.171,21.527,-42.872
C07961=1018.188,-0.510,-120.445,-24.171,21.526,-42.867
C07962=1018.187,-0.104,-120.479,-24.172,21.525,-42.862
C07963=1018.187,0.300,-120.513,-24.173,21.525,-42.857
C07964=1018.186,0.701,-120.547,-24.173,21.525,-42.851
C07965=1018.185,1.101,-120.582,-24.174,21.525,-42.846
C07966=1018.185,1.500,-120.615,-24.175,21.523,-42.841
C07967=1018.184,1.898,-120.648,-24.175,21.524,-42.836
C07968=1018.184,2.283,-120.681,-24.176,21.523,-42.833
C07969=1018.183,2.637,-120.711,-24.177,21.522,-42.827
C07970=1018.182,2.959,-120.738,-24.177,21.522,-42.823
C07971=1018.182,3.273,-120.765,-24.178,21.521,-42.817
C07972=1018.181,3.601,-120.793,-24.179,21.521,-42.812
C07973=1018.180,3.959,-120.823,-24.179,21.521,-42.809
C07974=1018.180,4.349,-120.856,-24.180,21.520,-42.805
C07975=1018.179,4.745,-120.890,-24.180,21.519,-42.799
C07976=1018.178,5.140,-120.924,-24.181,21.520,-42.794
C07977=1018.178,5.535,-120.957,-24.182,21.519,-42.790
C07978=1018.177,5.930,-120.991,-24.182,21.518,-42.785
C07979=1018.176,6.323,-121.024,-24.183,21.519,-42.779
C07980=1018.175,6.716,-121.058,-24.184,21.517,-42.775
C07981=1018.174,7.109,-121.091,-24.185,21.517,-42.770
C07982=1018.173,7.499,-121.125,-24.185,21.517,-42.764
C07983=1018.173,7.888,-121.158,-24.186,21.516,-42.761
C07984=1018.171,8.271,-121.190,-24.187,21.516,-42.755
C07985=1018.170,8.652,-121.223,-24.187,21.515,-42.751
C07986=1018.170,9.030,-121.255,-24.188,21.515,-42.746
C07987=1018.169,9.406,-121.288,-24.189,21.514,-42.740
C07988=1018.168,9.782,-121.320,-24.189,21.514,-42.737
C07989=1018.167,10.159,-121.352,-24.190,21.513,-42.731
C07990=1018.166,10.537,-121.385,-24.191,21.513,-42.726
C07991=1018.165,10.917,-121.417,-24.191,21.513,-42.722
C07992=1018.164,11.300,-121.450,-24.192,21.512,-42.716
C07993=1018.163,11.686,-121.483,-24.192,21.511,-42.713
C07994=1018.162,12.073,-121.516,-24.193,21.512,-42.707
C07995=1018.161,12.459,-121.549,-24.193,21.510,-42.703
C07996=1018.160,12.845,-121.582,-24.194,21.510,-42.698
C07997=1018.159,13.232,-121.616,-24.195,21.511,-42.693
C07998=1018.158,13.620,-121.649,-24.196,21.509,-42.689
C07999=1018.157,14.006,-121.683,-24.196,21.509,-42.683
C08000=1018.155,14.394,-121.716,-24.197,21.509,-42.680
C08001=1018.154,14.782,-121.749,-24.198,21.508,-42.674
C08002=1018.153,15.171,-121.783,-24.198,21.508,-42.670
C08003=1018.151,15.560,-121.816,-24.199,21.507,-42.665
C08004=1018.151,15.951,-121.850,-24.200,21.507,-42.659
C08005=1018.150,16.342,-121.884,-24.200,21.506,-42.656
C08006=1018.148,16.734,-121.917,-24.201,21.506,-42.650
C08007=1018.147,17.126,-121.952,-24.201,21.505,-42.646
C08008=1018.146,17.519,-121.985,-24.202,21.505,-42.641
C08009=1018.144,17.914,-122.019,-24.203,21.505,-42.635
C08010=1018.143,18.308,-122.054,-24.203,21.504,-42.632
C08011=1018.142,18.705,-122.088,-24.204,21.503,-42.626
C08012=1018.141,19.101,-122.123,-24.205,21.503,-42.622
C08013=1018.139,19.498,-122.157,-24.205,21.503,-42.617
C08014=1018.139,19.710,-122.175,-24.206,21.503,-42.613
C08015=1018.138,19.946,-122.195,-24.206,21.502,-42.610
C08016=1018.137,20.211,-122.219,-24.207,21.503,-42.606
C08017=1018.136,20.499,-122.244,-24.207,21.501,-42.604
C08018=1018.134,20.795,-122.270,-24.207,21.501,-42.602
C08019=1018.133,21.087,-122.295,-24.208,21.502,-42.599
C08020=1018.133,21.359,-122.318,-24.208,21.501,-42.597
C08021=1018.131,21.604,-122.339,-24.209,21.501,-42.593
C08022=1018.130,22.017,-122.376,-24.210,21.501,-42.586
C08023=1018.129,22.392,-122.409,-24.210,21.500,-42.584
C08024=1018.128,22.715,-122.436,-24.211,21.500,-42.580
C08025=1018.127,22.980,-122.459,-24.211,21.500,-42.577
C08026=1018.126,23.212,-122.479,-24.211,21.499,-42.573
C08027=1018.125,23.447,-122.500,-24.212,21.498,-42.567
C08028=1018.124,23.718,-122.524,-24.213,21.498,-42.564
C08029=1018.123,24.049,-122.552,-24.213,21.498,-42.562
C08030=1018.121,24.432,-122.585,-24.213,21.497,-42.558
C08031=1018.119,24.831,-122.620,-24.214,21.497,-42.553
C08032=1018.118,25.230,-122.655,-24.215,21.497,-42.549
C08033=1018.116,25.630,-122.690,-24.215,21.496,-42.543
C08034=1018.115,26.029,-122.725,-24.216,21.496,-42.540
C08035=1018.113,26.428,-122.760,-24.217,21.496,-42.534
C08036=1018.112,26.827,-122.795,-24.218,21.495,-42.529
C08037=1018.110,27.226,-122.830,-24.218,21.494,-42.525
C08038=1018.108,27.626,-122.865,-24.219,21.495,-42.520
C08039=1018.106,28.026,-122.900,-24.219,21.493,-42.516
C08040=1018.105,28.426,-122.935,-24.220,21.493,-42.510
C08041=1018.103,28.825,-122.970,-24.221,21.493,-42.507
C08042=1018.102,29.224,-123.005,-24.221,21.492,-42.501
C08043=1018.099,29.624,-123.040,-24.222,21.492,-42.497
C08044=1018.098,30.023,-123.075,-24.223,21.492,-42.492
C08045=1018.096,30.423,-123.109,-24.223,21.491,-42.488
C08046=1018.093,30.822,-123.145,-24.224,21.491,-42.483
C08047=1018.092,31.222,-123.180,-24.224,21.490,-42.479
C08048=1018.090,31.622,-123.216,-24.225,21.490,-42.474
C08049=1018.088,32.021,-123.251,-24.226,21.489,-42.469
C08050=1018.086,32.421,-123.286,-24.226,21.489,-42.464
C08051=1018.084,32.820,-123.320,-24.227,21.489,-42.461
C08052=1018.083,33.221,-123.356,-24.228,21.489,-42.455
C08053=1018.081,33.620,-123.391,-24.228,21.487,-42.451
C08054=1018.079,34.019,-123.427,-24.229,21.488,-42.446
C08055=1018.077,34.419,-123.462,-24.229,21.487,-42.442
C08056=1018.075,34.819,-123.497,-24.230,21.486,-42.437
C08057=1018.073,35.219,-123.532,-24.231,21.486,-42.433
C08058=1018.070,35.619,-123.568,-24.231,21.486,-42.428
C08059=1018.069,36.018,-123.603,-24.232,21.486,-42.424
C08060=1018.067,36.418,-123.639,-24.233,21.485,-42.418
C08061=1018.064,36.818,-123.674,-24.233,21.484,-42.414
C08062=1018.062,37.218,-123.709,-24.234,21.485,-42.409
C08063=1018.061,37.618,-123.744,-24.235,21.484,-42.405
C08064=1018.059,38.017,-123.780,-24.235,21.483,-42.400
C08065=1018.056,38.417,-123.816,-24.236,21.483,-42.396
C08066=1018.054,38.818,-123.851,-24.237,21.483,-42.391
C08067=1018.052,39.217,-123.886,-24.237,21.483,-42.387
C08068=1018.050,39.617,-123.922,-24.238,21.482,-42.383
C08069=1018.048,40.017,-123.958,-24.238,21.481,-42.378
C08070=1018.045,40.417,-123.992,-24.239,21.481,-42.374
C08071=1018.043,40.817,-124.028,-24.240,21.481,-42.369
C08072=1018.041,41.217,-124.064,-24.240,21.481,-42.365
C08073=1018.039,41.616,-124.099,-24.241,21.480,-42.359
C08074=1018.037,42.017,-124.135,-24.241,21.479,-42.356
C08075=1018.034,42.417,-124.171,-24.242,21.479,-42.352
C08076=1018.032,42.817,-124.206,-24.243,21.479,-42.347
C08077=1018.030,43.217,-124.242,-24.243,21.479,-42.343
C08078=1018.028,43.616,-124.278,-24.244,21.479,-42.338
C08079=1018.026,44.017,-124.313,-24.244,21.477,-42.333
C08080=1018.022,44.417,-124.349,-24.245,21.477,-42.330
C08081=1018.020,44.817,-124.384,-24.246,21.477,-42.325
C08082=1018.018,45.217,-124.420,-24.246,21.477,-42.321
C08083=1018.015,45.617,-124.456,-24.247,21.477,-42.316
C08084=1018.013,46.018,-124.492,-24.247,21.475,-42.311
C08085=1018.011,46.417,-124.527,-24.248,21.475,-42.308
C08086=1018.008,46.817,-124.563,-24.249,21.475,-42.302
C08087=1018.006,47.217,-124.599,-24.249,21.475,-42.299
C08088=1018.003,47.617,-124.635,-24.250,21.474,-42.295
C08089=1018.001,48.018,-124.670,-24.251,21.474,-42.290
C08090=1017.998,48.418,-124.707,-24.251,21.474,-42.286
C08091=1017.996,48.817,-124.742,-24.251,21.472,-42.282
C08092=1017.993,49.218,-124.779,-24.252,21.473,-42.277
C08093=1017.991,49.618,-124.813,-24.253,21.472,-42.273
C08094=1017.988,50.019,-124.850,-24.254,21.472,-42.268
C08095=1017.985,50.418,-124.886,-24.254,21.472,-42.264
C08096=1017.983,50.819,-124.922,-24.255,21.471,-42.260
C08097=1017.980,51.218,-124.958,-24.255,21.471,-42.255
C08098=1017.977,51.618,-124.994,-24.256,21.471,-42.251
C08099=1017.975,52.019,-125.029,-24.256,21.470,-42.247
C08100=1017.972,52.419,-125.065,-24.257,21.469,-42.243
C08101=1017.970,52.820,-125.102,-24.258,21.469,-42.238
C08102=1017.967,53.219,-125.138,-24.258,21.469,-42.234
C08103=1017.964,53.619,-125.174,-24.259,21.468,-42.230
C08104=1017.961,54.020,-125.209,-24.259,21.468,-42.225
C08105=1017.958,54.420,-125.245,-24.260,21.468,-42.221
C08106=1017.956,54.821,-125.282,-24.260,21.468,-42.218
C08107=1017.953,55.220,-125.318,-24.261,21.468,-42.212
C08108=1017.950,55.620,-125.354,-24.262,21.467,-42.209
C08109=1017.947,56.021,-125.391,-24.262,21.467,-42.205
C08110=1017.945,56.420,-125.426,-24.263,21.465,-42.201
C08111=1017.942,56.822,-125.462,-24.264,21.466,-42.196
C08112=1017.939,57.221,-125.498,-24.264,21.465,-42.192
C08113=1017.936,57.621,-125.534,-24.264,21.465,-42.188
C08114=1017.934,58.022,-125.571,-24.265,21.465,-42.183
C08115=1017.931,58.422,-125.607,-24.266,21.464,-42.179
C08116=1017.927,58.822,-125.644,-24.266,21.464,-42.175
C08117=1017.924,59.222,-125.680,-24.267,21.463,-42.172
C08118=1017.921,59.622,-125.716,-24.268,21.464,-42.166
C08119=1017.918,60.022,-125.752,-24.268,21.463,-42.163
C08120=1017.915,60.423,-125.788,-24.269,21.463,-42.159
C08121=1017.912,60.823,-125.824,-24.269,21.462,-42.155
C08122=1017.909,61.223,-125.860,-24.270,21.462,-42.150
C08123=1017.907,61.623,-125.897,-24.270,21.462,-42.146
C08124=1017.903,62.024,-125.933,-24.271,21.461,-42.142
C08125=1017.900,62.424,-125.970,-24.271,21.461,-42.139
C08126=1017.897,62.843,-126.008,-24.272,21.460,-42.133
C08127=1017.895,63.097,-126.031,-24.272,21.460,-42.131
C08128=1017.893,63.364,-126.055,-24.273,21.460,-42.129
C08129=1017.891,63.614,-126.078,-24.273,21.459,-42.127
C08130=1017.890,63.831,-126.097,-24.274,21.460,-42.124
C08131=1017.888,64.038,-126.116,-24.274,21.460,-42.122
C08132=1017.886,64.256,-126.136,-24.274,21.459,-42.120
C08133=1017.885,64.485,-126.157,-24.274,21.459,-42.116
C08134=1017.882,64.722,-126.179,-24.275,21.459,-42.115
C08135=1017.881,64.957,-126.200,-24.275,21.458,-42.113
C08136=1017.879,65.188,-126.221,-24.275,21.458,-42.111
C08137=1017.877,65.408,-126.241,-24.276,21.459,-42.108
C08138=1017.875,65.621,-126.261,-24.276,21.458,-42.106
C08139=1017.872,66.030,-126.297,-24.277,21.458,-42.102
C08140=1017.869,66.427,-126.334,-24.277,21.457,-42.098
C08141=1017.865,66.828,-126.370,-24.278,21.457,-42.094
C08142=1017.862,67.230,-126.407,-24.278,21.457,-42.089
C08143=1017.859,67.634,-126.444,-24.279,21.457,-42.085
C08144=1017.855,68.038,-126.481,-24.279,21.456,-42.082
C08145=1017.853,68.444,-126.518,-24.280,21.456,-42.078
C08146=1017.849,68.852,-126.556,-24.280,21.455,-42.074
C08147=1017.846,69.260,-126.592,-24.281,21.455,-42.069
C08148=1017.842,69.671,-126.630,-24.282,21.455,-42.065
C08149=1017.839,70.082,-126.667,-24.282,21.454,-42.061
C08150=1017.835,70.493,-126.705,-24.283,21.454,-42.058
C08151=1017.832,70.905,-126.742,-24.283,21.453,-42.054
C08152=1017.828,71.316,-126.780,-24.284,21.454,-42.049
C08153=1017.824,71.727,-126.818,-24.285,21.453,-42.045
C08154=1017.821,72.138,-126.856,-24.285,21.453,-42.041
C08155=1017.818,72.552,-126.893,-24.285,21.452,-42.037
C08156=1017.814,72.967,-126.932,-24.286,21.452,-42.034
C08157=1017.811,73.385,-126.970,-24.287,21.452,-42.028
C08158=1017.806,73.806,-127.008,-24.287,21.452,-42.025
C08159=1017.805,74.017,-127.028,-24.288,21.451,-42.023
C08160=1017.803,74.229,-127.047,-24.288,21.451,-42.021
C08161=1017.801,74.442,-127.066,-24.288,21.451,-42.019
C08162=1017.799,74.655,-127.087,-24.288,21.451,-42.017
C08163=1017.797,74.869,-127.106,-24.289,21.450,-42.015
C08164=1017.795,75.082,-127.126,-24.289,21.451,-42.012
C08165=1017.794,75.296,-127.145,-24.289,21.451,-42.010
C08166=1017.792,75.508,-127.164,-24.290,21.450,-42.008
C08167=1017.787,75.928,-127.203,-24.290,21.450,-42.004
C08168=1017.784,76.339,-127.241,-24.291,21.449,-42.001
C08169=1017.781,76.741,-127.278,-24.291,21.449,-41.997
C08170=1017.777,77.136,-127.314,-24.292,21.449,-41.994
C08171=1017.773,77.524,-127.350,-24.292,21.448,-41.989
C08172=1017.770,77.910,-127.385,-24.293,21.447,-41.986
C08173=1017.766,78.297,-127.421,-24.293,21.448,-41.980
C08174=1017.762,78.688,-127.457,-24.294,21.447,-41.977
C08175=1017.759,79.085,-127.493,-24.294,21.447,-41.973
C08176=1017.755,79.491,-127.531,-24.295,21.447,-41.970
C08177=1017.751,79.905,-127.569,-24.296,21.447,-41.966
C08178=1017.749,80.115,-127.588,-24.296,21.446,-41.964
C08179=1017.747,80.327,-127.608,-24.296,21.446,-41.962
C08180=1017.745,80.539,-127.628,-24.296,21.446,-41.960
C08181=1017.743,80.752,-127.647,-24.297,21.446,-41.958
C08182=1017.741,80.965,-127.667,-24.297,21.445,-41.956
C08183=1017.739,81.178,-127.687,-24.297,21.445,-41.955
C08184=1017.737,81.390,-127.706,-24.297,21.445,-41.953
C08185=1017.735,81.603,-127.726,-24.298,21.445,-41.951
C08186=1017.733,81.815,-127.745,-24.298,21.445,-41.949
C08187=1017.731,82.026,-127.765,-24.298,21.444,-41.947
C08188=1017.729,82.238,-127.784,-24.299,21.445,-41.944
C08189=1017.727,82.449,-127.804,-24.299,21.444,-41.942
C08190=1017.725,82.660,-127.823,-24.299,21.444,-41.940
C08191=1017.723,82.871,-127.842,-24.299,21.444,-41.938
C08192=1017.719,83.291,-127.881,-24.300,21.444,-41.935
C08193=1017.714,83.709,-127.920,-24.300,21.444,-41.931
C08194=1017.710,84.127,-127.958,-24.301,21.443,-41.927
C08195=1017.707,84.542,-127.997,-24.301,21.443,-41.923
C08196=1017.703,84.956,-128.035,-24.302,21.443,-41.920
C08197=1017.698,85.369,-128.073,-24.302,21.442,-41.916
C08198=1017.694,85.780,-128.111,-24.303,21.442,-41.912
C08199=1017.690,86.189,-128.149,-24.303,21.441,-41.908
C08200=1017.686,86.596,-128.188,-24.304,21.442,-41.905
C08201=1017.682,87.002,-128.225,-24.304,21.441,-41.901
C08202=1017.678,87.405,-128.262,-24.305,21.441,-41.898
C08203=1017.674,87.801,-128.299,-24.305,21.440,-41.894
C08204=1017.670,88.189,-128.334,-24.306,21.440,-41.890
C08205=1017.666,88.573,-128.370,-24.307,21.440,-41.887
C08206=1017.662,88.956,-128.405,-24.307,21.440,-41.883
C08207=1017.658,89.342,-128.442,-24.308,21.439,-41.879
C08208=1017.654,89.735,-128.477,-24.308,21.439,-41.875
C08209=1017.650,90.133,-128.515,-24.309,21.439,-41.872
C08210=1017.646,90.532,-128.552,-24.309,21.439,-41.868
C08211=1017.642,90.931,-128.589,-24.310,21.438,-41.865
C08212=1017.637,91.330,-128.626,-24.310,21.438,-41.861
C08213=1017.633,91.730,-128.664,-24.311,21.438,-41.857
C08214=1017.629,92.129,-128.701,-24.311,21.438,-41.854
C08215=1017.625,92.528,-128.737,-24.312,21.437,-41.850
C08216=1017.620,92.927,-128.775,-24.312,21.437,-41.846
C08217=1017.616,93.326,-128.812,-24.312,21.437,-41.844
C08218=1017.612,93.725,-128.849,-24.313,21.436,-41.841
C08219=1017.608,94.124,-128.886,-24.313,21.436,-41.837
C08220=1017.603,94.523,-128.924,-24.314,21.435,-41.833
C08221=1017.599,94.922,-128.961,-24.315,21.436,-41.830
C08222=1017.594,95.321,-128.997,-24.315,21.435,-41.826
C08223=1017.590,95.720,-129.034,-24.316,21.435,-41.822
C08224=1017.585,96.119,-129.072,-24.316,21.435,-41.819
C08225=1017.581,96.518,-129.109,-24.317,21.435,-41.815
C08226=1017.577,96.917,-129.146,-24.317,21.434,-41.811
C08227=1017.572,97.316,-129.184,-24.318,21.434,-41.808
C08228=1017.568,97.715,-129.221,-24.318,21.433,-41.806
C08229=1017.563,98.113,-129.258,-24.318,21.433,-41.802
C08230=1017.559,98.512,-129.295,-24.319,21.432,-41.798
C08231=1017.555,98.911,-129.332,-24.319,21.433,-41.795
C08232=1017.550,99.310,-129.370,-24.320,21.432,-41.791
C08233=1017.546,99.709,-129.407,-24.320,21.432,-41.787
C08234=1017.541,100.108,-129.444,-24.321,21.432,-41.784
C08235=1017.536,100.506,-129.481,-24.322,21.432,-41.780
C08236=1017.531,100.905,-129.519,-24.322,21.431,-41.778
C08237=1017.527,101.304,-129.556,-24.322,21.431,-41.775
C08238=1017.522,101.703,-129.593,-24.323,21.431,-41.771
C08239=1017.518,102.101,-129.630,-24.323,21.430,-41.767
C08240=1017.513,102.500,-129.668,-24.324,21.430,-41.763
C08241=1017.509,102.899,-129.705,-24.324,21.430,-41.760
C08242=1017.503,103.298,-129.742,-24.325,21.430,-41.756
C08243=1017.499,103.696,-129.780,-24.325,21.430,-41.754
C08244=1017.494,104.094,-129.817,-24.326,21.429,-41.751
C08245=1017.490,104.493,-129.854,-24.326,21.429,-41.747
C08246=1017.485,104.892,-129.892,-24.327,21.429,-41.743
C08247=1017.480,105.291,-129.929,-24.327,21.429,-41.740
C08248=1017.476,105.690,-129.966,-24.328,21.428,-41.736
C08249=1017.470,106.088,-130.004,-24.328,21.428,-41.734
C08250=1017.465,106.487,-130.041,-24.328,21.427,-41.730
C08251=1017.461,106.885,-130.078,-24.329,21.427,-41.727
C08252=1017.456,107.284,-130.116,-24.330,21.427,-41.723
C08253=1017.451,107.682,-130.154,-24.330,21.427,-41.719
C08254=1017.447,108.081,-130.191,-24.330,21.426,-41.717
C08255=1017.441,108.479,-130.228,-24.331,21.426,-41.714
C08256=1017.436,108.879,-130.266,-24.331,21.426,-41.710
C08257=1017.432,109.277,-130.302,-24.332,21.426,-41.707
C08258=1017.427,109.675,-130.341,-24.332,21.426,-41.703
C08259=1017.422,110.074,-130.378,-24.333,21.425,-41.701
C08260=1017.417,110.473,-130.416,-24.333,21.425,-41.697
C08261=1017.411,110.871,-130.453,-24.334,21.425,-41.694
C08262=1017.407,111.269,-130.490,-24.334,21.425,-41.690
C08263=1017.402,111.668,-130.527,-24.334,21.424,-41.688
C08264=1017.397,112.066,-130.565,-24.335,21.423,-41.684
C08265=1017.392,112.465,-130.603,-24.335,21.424,-41.681
C08266=1017.386,112.864,-130.640,-24.336,21.423,-41.677
C08267=1017.381,113.262,-130.678,-24.336,21.423,-41.675
C08268=1017.376,113.661,-130.715,-24.337,21.423,-41.671
C08269=1017.371,114.059,-130.753,-24.337,21.422,-41.668
C08270=1017.366,114.458,-130.791,-24.338,21.423,-41.664
C08271=1017.361,114.857,-130.828,-24.338,21.422,-41.662
C08272=1017.355,115.255,-130.865,-24.339,21.422,-41.659
C08273=1017.350,115.653,-130.903,-24.339,21.422,-41.655
C08274=1017.345,116.051,-130.941,-24.340,21.422,-41.652
C08275=1017.340,116.451,-130.978,-24.340,21.421,-41.649
C08276=1017.334,116.849,-131.016,-24.340,21.420,-41.646
C08277=1017.329,117.247,-131.053,-24.341,21.421,-41.642
C08278=1017.325,117.646,-131.091,-24.341,21.420,-41.638
C08279=1017.319,118.044,-131.129,-24.342,21.420,-41.637
C08280=1017.314,118.443,-131.166,-24.342,21.420,-41.633
C08281=1017.308,118.841,-131.203,-24.343,21.420,-41.629
C08282=1017.303,119.239,-131.241,-24.343,21.420,-41.626
C08283=1017.298,119.638,-131.280,-24.343,21.419,-41.624
C08284=1017.292,120.037,-131.317,-24.344,21.419,-41.620
C08285=1017.287,120.435,-131.354,-24.345,21.419,-41.617
C08286=1017.282,120.834,-131.392,-24.345,21.418,-41.614
C08287=1017.277,121.232,-131.430,-24.345,21.418,-41.611
C08288=1017.272,121.631,-131.468,-24.346,21.418,-41.607
C08289=1017.267,122.029,-131.505,-24.346,21.417,-41.605
C08290=1017.261,122.428,-131.544,-24.347,21.418,-41.602
C08291=1017.256,122.826,-131.582,-24.347,21.417,-41.598
C08292=1017.251,123.225,-131.620,-24.348,21.418,-41.595
C08293=1017.246,123.623,-131.657,-24.348,21.416,-41.592
C08294=1017.242,124.022,-131.696,-24.348,21.417,-41.589
C08295=1017.235,124.421,-131.734,-24.349,21.416,-41.585
C08296=1017.230,124.819,-131.771,-24.349,21.416,-41.583
C08297=1017.225,125.218,-131.809,-24.350,21.416,-41.580
C08298=1017.220,125.616,-131.847,-24.350,21.416,-41.576
C08299=1017.215,126.015,-131.886,-24.350,21.415,-41.574
C08300=1017.209,126.413,-131.923,-24.351,21.415,-41.571
C08301=1017.205,126.812,-131.961,-24.351,21.415,-41.567
C08302=1017.199,127.211,-131.999,-24.352,21.415,-41.565
C08303=1017.194,127.609,-132.037,-24.352,21.414,-41.561
C08304=1017.188,128.008,-132.075,-24.353,21.415,-41.558
C08305=1017.183,128.406,-132.113,-24.353,21.414,-41.555
C08306=1017.178,128.805,-132.151,-24.354,21.414,-41.552
C08307=1017.172,129.203,-132.190,-24.354,21.413,-41.550
C08308=1017.167,129.602,-132.227,-24.354,21.413,-41.547
C08309=1017.161,130.001,-132.265,-24.355,21.413,-41.543
C08310=1017.156,130.399,-132.304,-24.355,21.413,-41.541
C08311=1017.150,130.798,-132.341,-24.356,21.413,-41.538
C08312=1017.145,131.196,-132.379,-24.356,21.413,-41.534
C08313=1017.140,131.595,-132.418,-24.356,21.412,-41.532
C08314=1017.133,131.994,-132.456,-24.357,21.412,-41.528
C08315=1017.129,132.393,-132.494,-24.357,21.412,-41.525
C08316=1017.123,132.791,-132.532,-24.358,21.411,-41.523
C08317=1017.118,133.189,-132.570,-24.358,21.412,-41.519
C08318=1017.112,133.589,-132.608,-24.358,21.411,-41.517
C08319=1017.106,133.987,-132.646,-24.359,21.411,-41.514
C08320=1017.101,134.386,-132.685,-24.359,21.411,-41.510
C08321=1017.095,134.785,-132.722,-24.360,21.410,-41.508
C08322=1017.089,135.183,-132.760,-24.360,21.411,-41.505
C08323=1017.084,135.578,-132.798,-24.360,21.410,-41.502
C08324=1017.078,135.949,-132.834,-24.361,21.409,-41.500
C08325=1017.073,136.290,-132.866,-24.361,21.410,-41.497
C08326=1017.069,136.608,-132.897,-24.361,21.409,-41.495
C08327=1017.064,136.923,-132.927,-24.362,21.409,-41.491
C08328=1017.060,137.260,-132.960,-24.363,21.410,-41.488
C08329=1017.054,137.630,-132.995,-24.363,21.408,-41.486
C08330=1017.049,138.031,-133.033,-24.363,21.408,-41.484
C08331=1017.046,138.237,-133.053,-24.363,21.408,-41.482
C08332=1017.042,138.454,-133.074,-24.364,21.408,-41.480
C08333=1017.039,138.691,-133.097,-24.364,21.408,-41.478
C08334=1017.036,138.951,-133.121,-24.364,21.407,-41.476
C08335=1017.031,139.229,-133.148,-24.364,21.408,-41.475
C08336=1017.027,139.516,-133.175,-24.365,21.408,-41.473
C08337=1017.023,139.804,-133.203,-24.365,21.408,-41.471
C08338=1017.018,140.081,-133.230,-24.365,21.408,-41.470
C08339=1017.015,140.340,-133.254,-24.366,21.408,-41.468
C08340=1017.012,140.576,-133.277,-24.366,21.408,-41.466
C08341=1017.005,140.993,-133.317,-24.366,21.407,-41.462
C08342=1016.999,141.398,-133.356,-24.366,21.406,-41.460
C08343=1016.994,141.803,-133.395,-24.367,21.407,-41.457
C08344=1016.987,142.209,-133.433,-24.368,21.406,-41.453
C08345=1016.982,142.616,-133.473,-24.368,21.406,-41.451
C08346=1016.975,143.024,-133.512,-24.368,21.406,-41.448
C08347=1016.969,143.433,-133.551,-24.369,21.405,-41.445
C08348=1016.963,143.842,-133.590,-24.369,21.406,-41.442
C08349=1016.956,144.252,-133.630,-24.370,21.405,-41.438
C08350=1016.950,144.664,-133.670,-24.370,21.405,-41.436
C08351=1016.943,145.075,-133.709,-24.370,21.405,-41.432
C08352=1016.937,145.487,-133.748,-24.371,21.404,-41.431
C08353=1016.932,145.900,-133.787,-24.371,21.405,-41.427
C08354=1016.925,146.312,-133.827,-24.372,21.404,-41.424
C08355=1016.918,146.726,-133.867,-24.372,21.404,-41.422
C08356=1016.912,147.139,-133.907,-24.372,21.404,-41.418
C08357=1016.905,147.552,-133.947,-24.373,21.403,-41.416
C08358=1016.899,147.966,-133.987,-24.373,21.403,-41.412
C08359=1016.893,148.381,-134.026,-24.374,21.403,-41.409
C08360=1016.886,148.794,-134.066,-24.374,21.403,-41.407
C08361=1016.880,149.208,-134.106,-24.375,21.403,-41.403
C08362=1016.874,149.623,-134.145,-24.375,21.402,-41.401
C08363=1016.866,150.036,-134.185,-24.375,21.402,-41.398
C08364=1016.861,150.451,-134.225,-24.376,21.402,-41.394
C08365=1016.854,150.864,-134.265,-24.376,21.401,-41.392
C08366=1016.848,151.278,-134.305,-24.377,21.402,-41.389
C08367=1016.841,151.691,-134.345,-24.377,21.402,-41.387
C08368=1016.834,152.104,-134.384,-24.377,21.401,-41.383
C08369=1016.827,152.517,-134.424,-24.378,21.401,-41.381
C08370=1016.820,152.929,-134.464,-24.378,21.400,-41.377
C08371=1016.814,153.341,-134.503,-24.378,21.400,-41.375
C08372=1016.808,153.752,-134.542,-24.379,21.401,-41.372
C08373=1016.801,154.162,-134.582,-24.380,21.400,-41.368
C08374=1016.794,154.572,-134.622,-24.380,21.400,-41.366
C08375=1016.787,154.982,-134.661,-24.380,21.400,-41.363
C08376=1016.781,155.390,-134.700,-24.381,21.399,-41.361
C08377=1016.774,155.798,-134.740,-24.381,21.400,-41.358
C08378=1016.767,156.204,-134.779,-24.381,21.399,-41.355
C08379=1016.761,156.611,-134.818,-24.382,21.399,-41.352
C08380=1016.754,157.015,-134.857,-24.382,21.399,-41.350
C08381=1016.747,157.419,-134.896,-24.383,21.398,-41.346
C08382=1016.740,157.824,-134.935,-24.383,21.398,-41.344
C08383=1016.733,158.226,-134.973,-24.383,21.399,-41.341
C08384=1016.727,158.628,-135.013,-24.384,21.397,-41.339
C08385=1016.720,159.028,-135.051,-24.384,21.398,-41.335
C08386=1016.713,159.429,-135.090,-24.384,21.398,-41.333
C08387=1016.709,159.829,-135.129,-24.385,21.397,-41.330
C08388=1016.708,160.226,-135.171,-24.385,21.397,-41.328
C08389=1016.706,160.632,-135.214,-24.386,21.397,-41.325
C08390=1016.705,160.844,-135.236,-24.386,21.397,-41.324
C08391=1016.704,161.069,-135.259,-24.386,21.396,-41.322
C08392=1016.703,161.307,-135.284,-24.386,21.396,-41.320
C08393=1016.703,161.558,-135.310,-24.387,21.397,-41.319
C08394=1016.702,161.820,-135.338,-24.387,21.397,-41.317
C08395=1016.700,162.089,-135.366,-24.387,21.396,-41.315
C08396=1016.699,162.361,-135.394,-24.387,21.396,-41.313
C08397=1016.699,162.629,-135.423,-24.388,21.396,-41.311
C08398=1016.698,162.892,-135.450,-24.388,21.396,-41.309
C08399=1016.697,163.147,-135.476,-24.388,21.395,-41.308
C08400=1016.696,163.382,-135.502,-24.388,21.396,-41.306
C08401=1016.695,163.794,-135.545,-24.389,21.395,-41.304
C08402=1016.694,163.984,-135.565,-24.389,21.395,-41.302
C08403=1016.693,164.371,-135.605,-24.389,21.395,-41.300
C08404=1016.692,164.770,-135.647,-24.390,21.395,-41.297
C08405=1016.690,165.170,-135.690,-24.390,21.395,-41.295
C08406=1016.689,165.571,-135.732,-24.390,21.394,-41.291
C08407=1016.687,165.971,-135.774,-24.391,21.394,-41.289
C08408=1016.686,166.371,-135.816,-24.391,21.395,-41.286
C08409=1016.684,166.772,-135.859,-24.391,21.393,-41.284
C08410=1016.683,167.172,-135.900,-24.392,21.394,-41.280
C08411=1016.682,167.572,-135.943,-24.392,21.394,-41.278
C08412=1016.681,167.973,-135.985,-24.393,21.394,-41.275
C08413=1016.679,168.373,-136.027,-24.393,21.393,-41.273
C08414=1016.677,168.774,-136.069,-24.393,21.393,-41.271
C08415=1016.676,169.174,-136.112,-24.394,21.393,-41.267
C08416=1016.675,169.575,-136.154,-24.394,21.392,-41.265
C08417=1016.674,169.975,-136.196,-24.395,21.392,-41.262
C08418=1016.672,170.376,-136.238,-24.395,21.392,-41.260
C08419=1016.671,170.777,-136.281,-24.395,21.392,-41.256
C08420=1016.670,171.177,-136.323,-24.396,21.392,-41.254
C08421=1016.668,171.578,-136.366,-24.396,21.392,-41.251
C08422=1016.667,171.978,-136.409,-24.396,21.392,-41.249
C08423=1016.666,172.379,-136.450,-24.397,21.391,-41.247
C08424=1016.665,172.780,-136.493,-24.397,21.391,-41.243
C08425=1016.663,173.180,-136.536,-24.397,21.391,-41.242
C08426=1016.662,173.581,-136.578,-24.398,21.390,-41.238
C08427=1016.661,173.982,-136.621,-24.398,21.390,-41.236
C08428=1016.660,174.382,-136.664,-24.399,21.391,-41.233
C08429=1016.658,174.783,-136.706,-24.399,21.390,-41.231
C08430=1016.657,175.184,-136.749,-24.400,21.390,-41.227
C08431=1016.656,175.584,-136.791,-24.400,21.390,-41.225
C08432=1016.654,175.985,-136.833,-24.400,21.390,-41.223
C08433=1016.653,176.385,-136.876,-24.401,21.389,-41.219
C08434=1016.652,176.786,-136.919,-24.401,21.389,-41.218
C08435=1016.650,177.187,-136.962,-24.401,21.389,-41.214
C08436=1016.649,177.588,-137.005,-24.402,21.389,-41.212
C08437=1016.649,177.989,-137.047,-24.402,21.389,-41.209
C08438=1016.647,178.390,-137.090,-24.402,21.388,-41.207
C08439=1016.646,178.790,-137.132,-24.403,21.388,-41.205
C08440=1016.645,179.191,-137.176,-24.403,21.388,-41.201
C08441=1016.644,179.592,-137.219,-24.403,21.388,-41.199
C08442=1016.642,179.993,-137.261,-24.404,21.388,-41.196
C08443=1016.641,180.394,-137.304,-24.404,21.388,-41.194
C08444=1016.640,180.795,-137.347,-24.405,21.387,-41.190
C08445=1016.639,181.195,-137.390,-24.405,21.387,-41.188
C08446=1016.638,181.596,-137.433,-24.405,21.387,-41.186
C08447=1016.636,181.998,-137.476,-24.406,21.387,-41.183
C08448=1016.635,182.399,-137.519,-24.406,21.386,-41.181
C08449=1016.634,182.799,-137.562,-24.407,21.387,-41.177
C08450=1016.633,183.199,-137.604,-24.407,21.386,-41.176
C08451=1016.632,183.601,-137.648,-24.407,21.386,-41.172
C08452=1016.631,184.002,-137.691,-24.408,21.386,-41.170
C08453=1016.630,184.403,-137.734,-24.408,21.386,-41.168
C08454=1016.629,184.804,-137.778,-24.409,21.386,-41.165
C08455=1016.627,185.205,-137.820,-24.409,21.385,-41.162
C08456=1016.627,185.606,-137.863,-24.409,21.385,-41.159
C08457=1016.625,186.007,-137.906,-24.410,21.385,-41.157
C08458=1016.625,186.408,-137.950,-24.410,21.384,-41.155
C08459=1016.624,186.809,-137.993,-24.410,21.384,-41.151
C08460=1016.623,187.210,-138.036,-24.411,21.384,-41.150
C08461=1016.622,187.611,-138.079,-24.411,21.385,-41.146
C08462=1016.621,188.012,-138.123,-24.411,21.384,-41.144
C08463=1016.620,188.413,-138.165,-24.412,21.384,-41.141
C08464=1016.619,188.814,-138.209,-24.412,21.384,-41.139
C08465=1016.618,189.215,-138.252,-24.412,21.384,-41.137
C08466=1016.617,189.616,-138.295,-24.413,21.383,-41.133
C08467=1016.615,190.017,-138.339,-24.413,21.383,-41.131
C08468=1016.615,190.418,-138.383,-24.414,21.383,-41.128
C08469=1016.614,190.819,-138.426,-24.414,21.383,-41.126
C08470=1016.613,191.220,-138.470,-24.414,21.382,-41.124
C08471=1016.613,191.621,-138.513,-24.415,21.382,-41.120
C08472=1016.612,192.023,-138.556,-24.415,21.382,-41.118
C08473=1016.611,192.424,-138.600,-24.415,21.382,-41.115
C08474=1016.609,192.825,-138.643,-24.416,21.382,-41.113
C08475=1016.609,193.225,-138.687,-24.416,21.382,-41.109
C08476=1016.608,193.626,-138.730,-24.417,21.382,-41.108
C08477=1016.607,194.028,-138.774,-24.417,21.381,-41.105
C08478=1016.606,194.429,-138.817,-24.417,21.381,-41.102
C08479=1016.605,194.830,-138.862,-24.418,21.381,-41.100
C08480=1016.604,195.231,-138.905,-24.418,21.381,-41.097
C08481=1016.604,195.632,-138.948,-24.418,21.380,-41.094
C08482=1016.603,196.033,-138.992,-24.419,21.381,-41.091
C08483=1016.603,196.435,-139.036,-24.419,21.380,-41.089
C08484=1016.602,196.836,-139.080,-24.419,21.380,-41.087
C08485=1016.601,197.237,-139.123,-24.420,21.380,-41.084
C08486=1016.600,197.638,-139.167,-24.420,21.380,-41.082
C08487=1016.600,198.039,-139.211,-24.421,21.380,-41.078
C08488=1016.598,198.440,-139.255,-24.421,21.379,-41.076
C08489=1016.598,198.841,-139.299,-24.421,21.379,-41.074
C08490=1016.597,199.240,-139.342,-24.422,21.379,-41.071
C08491=1016.597,199.629,-139.385,-24.422,21.379,-41.069
C08492=1016.596,200.029,-139.429,-24.423,21.378,-41.065
C08493=1016.596,200.242,-139.452,-24.423,21.378,-41.065
C08494=1016.595,200.464,-139.476,-24.423,21.378,-41.063
C08495=1016.595,200.694,-139.502,-24.423,21.378,-41.061
C08496=1016.594,200.921,-139.527,-24.423,21.379,-41.060
C08497=1016.594,201.329,-139.571,-24.424,21.378,-41.058
C08498=1016.593,201.680,-139.610,-24.424,21.378,-41.054
C08499=1016.593,202.029,-139.648,-24.424,21.378,-41.052
C08500=1016.595,202.417,-139.692,-24.425,21.378,-41.051
C08501=1016.599,203.633,-139.827,-24.373,21.403,-41.416
C08502=1016.602,203.881,-139.855,-24.373,21.404,-41.415
C08503=1016.603,204.130,-139.882,-24.373,21.403,-41.414
C08504=1016.605,204.378,-139.909,-24.373,21.403,-41.412
C08505=1016.607,204.627,-139.936,-24.374,21.404,-41.411
C08506=1016.609,204.875,-139.965,-24.373,21.403,-41.410
C08507=1016.611,205.123,-139.991,-24.374,21.403,-41.409
C08508=1016.613,205.372,-140.018,-24.374,21.403,-41.407
C08509=1016.615,205.621,-140.046,-24.374,21.402,-41.407
C08510=1016.617,205.869,-140.074,-24.374,21.403,-41.405
C08511=1016.618,206.118,-140.102,-24.375,21.403,-41.403
C08512=1016.620,206.366,-140.129,-24.375,21.402,-41.401
C08513=1016.623,206.614,-140.156,-24.375,21.402,-41.401
C08514=1016.624,206.863,-140.184,-24.375,21.402,-41.399
C08515=1016.626,207.112,-140.211,-24.375,21.402,-41.398
C08516=1016.628,207.360,-140.239,-24.375,21.402,-41.398
C08517=1016.630,207.608,-140.266,-24.376,21.402,-41.396
C08518=1016.632,207.857,-140.293,-24.376,21.402,-41.394
C08519=1016.634,208.105,-140.322,-24.376,21.402,-41.392
C08520=1016.636,208.348,-140.348,-24.376,21.401,-41.392
C08521=1016.638,208.591,-140.375,-24.376,21.402,-41.391
C08522=1016.640,208.833,-140.402,-24.377,21.402,-41.389
C08523=1016.642,209.076,-140.428,-24.377,21.401,-41.388
C08524=1016.643,209.319,-140.456,-24.377,21.402,-41.387
C08525=1016.645,209.562,-140.483,-24.377,21.401,-41.385
C08526=1016.648,209.804,-140.510,-24.377,21.401,-41.383
C08527=1016.650,210.046,-140.537,-24.377,21.401,-41.383
C08528=1016.651,210.295,-140.564,-24.378,21.401,-41.381
C08529=1016.654,210.544,-140.592,-24.378,21.401,-41.379
C08530=1016.656,210.792,-140.619,-24.378,21.401,-41.378
C08531=1016.657,211.041,-140.647,-24.378,21.400,-41.377
C08532=1016.660,211.289,-140.675,-24.378,21.400,-41.375
C08533=1016.661,211.538,-140.702,-24.379,21.401,-41.374
C08534=1016.664,211.786,-140.730,-24.379,21.401,-41.372
C08535=1016.666,212.035,-140.757,-24.379,21.400,-41.372
C08536=1016.668,212.283,-140.786,-24.379,21.400,-41.370
C08537=1016.670,212.531,-140.813,-24.380,21.400,-41.368
C08538=1016.673,212.780,-140.841,-24.380,21.400,-41.366
C08539=1016.674,213.028,-140.869,-24.380,21.400,-41.366
C08540=1016.676,213.277,-140.896,-24.380,21.400,-41.365
C08541=1016.678,213.525,-140.924,-24.380,21.400,-41.363
C08542=1016.680,213.774,-140.952,-24.381,21.400,-41.361
C08543=1016.683,214.022,-140.979,-24.381,21.400,-41.359
C08544=1016.684,214.270,-141.008,-24.381,21.399,-41.359
C08545=1016.686,214.519,-141.035,-24.381,21.399,-41.357
C08546=1016.689,214.768,-141.063,-24.381,21.400,-41.356
C08547=1016.691,215.016,-141.090,-24.382,21.399,-41.354
C08548=1016.693,215.259,-141.117,-24.382,21.398,-41.353
C08549=1016.695,215.501,-141.145,-24.382,21.399,-41.352
C08550=1016.697,215.744,-141.172,-24.382,21.399,-41.350
C08551=1016.699,215.987,-141.199,-24.382,21.399,-41.348
C08552=1016.702,216.230,-141.226,-24.383,21.398,-41.346
C08553=1016.704,216.472,-141.253,-24.383,21.398,-41.346
C08554=1016.706,216.715,-141.281,-24.383,21.398,-41.344
C08555=1016.708,216.957,-141.308,-24.383,21.398,-41.342
C08556=1016.711,217.207,-141.335,-24.383,21.399,-41.341
C08557=1016.712,217.455,-141.364,-24.384,21.398,-41.339
C08558=1016.714,217.703,-141.391,-24.384,21.397,-41.339
C08559=1016.717,217.951,-141.420,-24.384,21.397,-41.337
C08560=1016.719,218.200,-141.447,-24.384,21.398,-41.335
C08561=1016.721,218.448,-141.475,-24.384,21.398,-41.333
C08562=1016.723,218.697,-141.503,-24.385,21.397,-41.332
C08563=1016.726,218.945,-141.531,-24.385,21.397,-41.330
C08564=1016.728,219.194,-141.559,-24.385,21.397,-41.330
C08565=1016.730,219.442,-141.587,-24.385,21.397,-41.328
C08566=1016.732,219.690,-141.615,-24.385,21.397,-41.326
C08567=1016.735,219.939,-141.643,-24.386,21.397,-41.324
C08568=1016.737,220.187,-141.671,-24.386,21.397,-41.323
C08569=1016.740,220.436,-141.699,-24.386,21.397,-41.321
C08570=1016.741,220.684,-141.727,-24.386,21.396,-41.320
C08571=1016.744,220.933,-141.755,-24.386,21.396,-41.318
C08572=1016.746,221.181,-141.782,-24.387,21.397,-41.317
C08573=1016.749,221.430,-141.811,-24.387,21.396,-41.315
C08574=1016.751,221.678,-141.839,-24.387,21.396,-41.313
C08575=1016.754,221.926,-141.867,-24.388,21.396,-41.311
C08576=1016.756,222.169,-141.895,-24.388,21.397,-41.310
C08577=1016.758,222.412,-141.922,-24.388,21.396,-41.309
C08578=1016.761,222.655,-141.949,-24.388,21.395,-41.308
C08579=1016.763,222.898,-141.977,-24.388,21.395,-41.306
C08580=1016.765,223.140,-142.004,-24.389,21.396,-41.304
C08581=1016.768,223.383,-142.032,-24.389,21.396,-41.302
C08582=1016.770,223.626,-142.060,-24.389,21.395,-41.300
C08583=1016.772,223.869,-142.086,-24.389,21.395,-41.300
C08584=1016.775,224.117,-142.115,-24.389,21.394,-41.298
C08585=1016.776,224.366,-142.143,-24.390,21.395,-41.297
C08586=1016.779,224.614,-142.171,-24.390,21.395,-41.295
C08587=1016.782,224.863,-142.199,-24.390,21.395,-41.293
C08588=1016.784,225.111,-142.228,-24.390,21.394,-41.291
C08589=1016.787,225.360,-142.256,-24.391,21.394,-41.289
C08590=1016.789,225.607,-142.283,-24.391,21.395,-41.288
C08591=1016.792,225.856,-142.312,-24.391,21.395,-41.286
C08592=1016.794,226.104,-142.340,-24.391,21.394,-41.285
C08593=1016.796,226.353,-142.368,-24.391,21.393,-41.284
C08594=1016.799,226.602,-142.396,-24.392,21.393,-41.282
C08595=1016.801,226.850,-142.424,-24.392,21.394,-41.280
C08596=1016.804,227.075,-142.450,-24.392,21.394,-41.278
C08597=1016.806,227.298,-142.476,-24.393,21.393,-41.276
C08598=1016.808,227.522,-142.501,-24.393,21.393,-41.275
C08599=1016.810,227.747,-142.527,-24.393,21.394,-41.273
C08600=1016.813,227.971,-142.553,-24.393,21.393,-41.273
C08601=1016.815,228.195,-142.578,-24.393,21.393,-41.271
C08602=1016.817,228.419,-142.603,-24.394,21.392,-41.269
C08603=1016.819,228.644,-142.629,-24.394,21.393,-41.267
C08604=1016.822,228.891,-142.657,-24.394,21.393,-41.266
C08605=1016.824,229.140,-142.686,-24.394,21.393,-41.264
C08606=1016.827,229.389,-142.714,-24.395,21.392,-41.262
C08607=1016.830,229.637,-142.742,-24.395,21.392,-41.260
C08608=1016.833,229.923,-142.775,-24.395,21.392,-41.258
C08609=1016.836,230.209,-142.807,-24.395,21.392,-41.256
C08610=1016.838,230.494,-142.840,-24.396,21.392,-41.254
C08611=1016.842,230.781,-142.873,-24.396,21.391,-41.252
C08612=1016.844,231.029,-142.901,-24.396,21.392,-41.251
C08613=1016.847,231.277,-142.929,-24.396,21.392,-41.249
C08614=1016.849,231.526,-142.958,-24.397,21.392,-41.247
C08615=1016.852,231.774,-142.987,-24.397,21.391,-41.245
C08616=1016.855,232.022,-143.014,-24.397,21.391,-41.243
C08617=1016.857,232.271,-143.043,-24.397,21.391,-41.242
C08618=1016.860,232.519,-143.072,-24.398,21.391,-41.240
C08619=1016.862,232.768,-143.101,-24.398,21.390,-41.238
C08620=1016.866,233.016,-143.129,-24.398,21.391,-41.236
C08621=1016.869,233.265,-143.157,-24.399,21.391,-41.234
C08622=1016.870,233.513,-143.186,-24.399,21.391,-41.233
C08623=1016.874,233.761,-143.214,-24.399,21.390,-41.231
C08624=1016.876,234.010,-143.243,-24.399,21.390,-41.229
C08625=1016.879,234.258,-143.271,-24.400,21.390,-41.227
C08626=1016.882,234.506,-143.300,-24.400,21.390,-41.225
C08627=1016.884,234.755,-143.329,-24.400,21.390,-41.223
C08628=1016.887,235.003,-143.357,-24.400,21.389,-41.221
C08629=1016.890,235.251,-143.385,-24.401,21.389,-41.219
C08630=1016.892,235.499,-143.415,-24.401,21.389,-41.218
C08631=1016.895,235.748,-143.443,-24.401,21.390,-41.216
C08632=1016.898,235.991,-143.471,-24.401,21.389,-41.214
C08633=1016.901,236.234,-143.499,-24.402,21.389,-41.212
C08634=1016.903,236.477,-143.527,-24.402,21.389,-41.210
C08635=1016.906,236.720,-143.555,-24.402,21.389,-41.209
C08636=1016.909,236.963,-143.583,-24.402,21.388,-41.207
C08637=1016.911,237.207,-143.611,-24.403,21.388,-41.205
C08638=1016.915,237.449,-143.639,-24.403,21.388,-41.203
C08639=1016.917,237.693,-143.668,-24.403,21.388,-41.201
C08640=1016.920,237.941,-143.696,-24.403,21.388,-41.199
C08641=1016.923,238.190,-143.724,-24.404,21.387,-41.197
C08642=1016.926,238.438,-143.754,-24.404,21.387,-41.195
C08643=1016.929,238.686,-143.783,-24.405,21.388,-41.192
C08644=1016.931,238.935,-143.811,-24.405,21.387,-41.190
C08645=1016.934,239.183,-143.840,-24.405,21.387,-41.188
C08646=1016.936,239.431,-143.868,-24.405,21.387,-41.186
C08647=1016.940,239.680,-143.897,-24.406,21.387,-41.184
C08648=1016.943,239.928,-143.926,-24.406,21.386,-41.183
C08649=1016.946,240.176,-143.956,-24.406,21.386,-41.181
C08650=1016.949,240.424,-143.984,-24.406,21.386,-41.179
C08651=1016.951,240.673,-144.013,-24.407,21.386,-41.177
C08652=1016.954,240.921,-144.042,-24.407,21.386,-41.174
C08653=1016.957,241.169,-144.070,-24.407,21.386,-41.172
C08654=1016.960,241.418,-144.099,-24.408,21.386,-41.170
C08655=1016.963,241.665,-144.128,-24.408,21.386,-41.168
C08656=1016.966,241.914,-144.157,-24.408,21.385,-41.166
C08657=1016.969,242.162,-144.185,-24.408,21.385,-41.164
C08658=1016.971,242.411,-144.215,-24.409,21.385,-41.162
C08659=1016.975,242.659,-144.244,-24.409,21.385,-41.159
C08660=1016.978,242.902,-144.272,-24.410,21.385,-41.157
C08661=1016.981,243.145,-144.300,-24.410,21.385,-41.155
C08662=1016.984,243.388,-144.329,-24.410,21.385,-41.153
C08663=1016.986,243.632,-144.357,-24.410,21.384,-41.151
C08664=1016.989,243.875,-144.386,-24.411,21.384,-41.150
C08665=1016.993,244.118,-144.414,-24.411,21.384,-41.148
C08666=1016.995,244.361,-144.443,-24.411,21.384,-41.144
C08667=1016.998,244.604,-144.471,-24.412,21.384,-41.143
C08668=1017.001,244.853,-144.501,-24.412,21.384,-41.141
C08669=1017.004,245.101,-144.529,-24.412,21.384,-41.139
C08670=1017.008,245.349,-144.558,-24.412,21.384,-41.137
C08671=1017.010,245.597,-144.587,-24.413,21.384,-41.134
C08672=1017.014,245.846,-144.617,-24.413,21.384,-41.132
C08673=1017.017,246.094,-144.646,-24.413,21.383,-41.129
C08674=1017.020,246.342,-144.675,-24.414,21.382,-41.127
C08675=1017.022,246.591,-144.703,-24.414,21.382,-41.126
C08676=1017.025,246.839,-144.732,-24.414,21.383,-41.122
C08677=1017.029,247.088,-144.761,-24.415,21.382,-41.120
C08678=1017.032,247.336,-144.791,-24.415,21.382,-41.118
C08679=1017.035,247.584,-144.820,-24.415,21.382,-41.117
C08680=1017.038,247.832,-144.850,-24.416,21.382,-41.113
C08681=1017.042,248.080,-144.879,-24.416,21.382,-41.111
C08682=1017.044,248.329,-144.908,-24.416,21.381,-41.109
C08683=1017.047,248.577,-144.937,-24.417,21.381,-41.107
C08684=1017.051,248.826,-144.967,-24.417,21.381,-41.104
C08685=1017.054,249.073,-144.995,-24.417,21.381,-41.102
C08686=1017.057,249.321,-145.024,-24.418,21.381,-41.100
C08687=1017.060,249.570,-145.054,-24.418,21.381,-41.098
C08688=1017.063,249.813,-145.083,-24.418,21.381,-41.095
C08689=1017.067,250.057,-145.111,-24.419,21.381,-41.093
C08690=1017.069,250.300,-145.140,-24.419,21.380,-41.091
C08691=1017.073,250.543,-145.169,-24.419,21.380,-41.089
C08692=1017.076,250.787,-145.197,-24.420,21.380,-41.085
C08693=1017.078,251.030,-145.226,-24.420,21.380,-41.084
C08694=1017.082,251.273,-145.255,-24.420,21.380,-41.082
C08695=1017.085,251.517,-145.284,-24.421,21.380,-41.078
C08696=1017.089,251.765,-145.313,-24.421,21.380,-41.076
C08697=1017.092,252.013,-145.343,-24.421,21.379,-41.074
C08698=1017.095,252.261,-145.372,-24.421,21.378,-41.072
C08699=1017.098,252.510,-145.402,-24.422,21.379,-41.069
C08700=1017.102,252.758,-145.431,-24.422,21.379,-41.067
C08701=1017.105,253.006,-145.461,-24.423,21.378,-41.065
C08702=1017.108,253.254,-145.490,-24.423,21.378,-41.061
C08703=1017.111,253.503,-145.519,-24.423,21.378,-41.060
C08704=1017.115,253.750,-145.549,-24.424,21.378,-41.058
C08705=1017.118,253.999,-145.578,-24.424,21.378,-41.054
C08706=1017.121,254.247,-145.607,-24.424,21.378,-41.052
C08707=1017.125,254.495,-145.637,-24.425,21.377,-41.049
C08708=1017.128,254.744,-145.667,-24.425,21.377,-41.047
C08709=1017.132,254.992,-145.697,-24.425,21.377,-41.045
C08710=1017.134,255.240,-145.726,-24.426,21.377,-41.042
C08711=1017.138,255.489,-145.755,-24.426,21.377,-41.040
C08712=1017.141,255.736,-145.785,-24.426,21.376,-41.037
C08713=1017.145,255.985,-145.814,-24.427,21.376,-41.034
C08714=1017.148,256.233,-145.845,-24.427,21.376,-41.032
C08715=1017.152,256.481,-145.874,-24.428,21.377,-41.029
C08716=1017.155,256.725,-145.903,-24.428,21.376,-41.027
C08717=1017.158,256.968,-145.933,-24.428,21.375,-41.025
C08718=1017.161,257.211,-145.962,-24.429,21.376,-41.021
C08719=1017.165,257.455,-145.991,-24.429,21.376,-41.019
C08720=1017.168,257.698,-146.020,-24.429,21.375,-41.018
C08721=1017.171,257.942,-146.049,-24.430,21.375,-41.014
C08722=1017.175,258.185,-146.078,-24.430,21.375,-41.012
C08723=1017.192,259.421,-146.232,-24.551,21.322,-40.171
C08724=1017.194,259.701,-146.268,-24.587,21.310,-39.930
C08725=1017.197,259.980,-146.305,-24.622,21.298,-39.688
C08726=1017.198,260.260,-146.343,-24.658,21.287,-39.446
C08727=1017.200,260.540,-146.381,-24.693,21.275,-39.204
C08728=1017.201,260.787,-146.416,-24.725,21.267,-38.988
C08729=1017.201,261.035,-146.451,-24.758,21.259,-38.770
C08730=1017.201,261.282,-146.486,-24.790,21.251,-38.554
C08731=1017.200,261.530,-146.522,-24.823,21.245,-38.337
C08732=1017.199,261.810,-146.564,-24.860,21.238,-38.090
C08733=1017.198,262.088,-146.606,-24.897,21.233,-37.842
C08734=1017.197,262.367,-146.649,-24.935,21.227,-37.593
C08735=1017.194,262.647,-146.692,-24.973,21.223,-37.345
C08736=1017.192,262.894,-146.731,-25.006,21.220,-37.124
C08737=1017.190,263.141,-146.770,-25.040,21.217,-36.903
C08738=1017.187,263.388,-146.810,-25.074,21.216,-36.681
C08739=1017.184,263.635,-146.850,-25.108,21.215,-36.458
C08740=1017.179,263.914,-146.897,-25.147,21.216,-36.205
C08741=1017.174,264.193,-146.944,-25.186,21.217,-35.952
C08742=1017.169,264.472,-146.991,-25.226,21.219,-35.699
C08743=1017.164,264.751,-147.040,-25.265,21.221,-35.444
C08744=1017.158,264.997,-147.084,-25.300,21.225,-35.219
C08745=1017.153,265.243,-147.127,-25.335,21.229,-34.991
C08746=1017.146,265.489,-147.171,-25.370,21.233,-34.766
C08747=1017.140,265.735,-147.216,-25.406,21.239,-34.538
C08748=1017.133,266.015,-147.267,-25.446,21.246,-34.279
C08749=1017.125,266.293,-147.319,-25.487,21.254,-34.021
C08750=1017.116,266.572,-147.372,-25.527,21.264,-33.760
C08751=1017.107,266.851,-147.426,-25.568,21.275,-33.499
C08752=1017.099,267.096,-147.473,-25.604,21.284,-33.269
C08753=1017.090,267.341,-147.522,-25.641,21.295,-33.037
C08754=1017.081,267.586,-147.571,-25.677,21.306,-32.805
C08755=1017.071,267.831,-147.619,-25.713,21.318,-32.573
C08756=1017.060,268.110,-147.676,-25.755,21.333,-32.307
C08757=1017.048,268.388,-147.733,-25.797,21.350,-32.039
C08758=1017.036,268.667,-147.791,-25.839,21.367,-31.772
C08759=1017.023,268.945,-147.850,-25.881,21.386,-31.502
C08760=1017.012,269.190,-147.901,-25.918,21.402,-31.266
C08761=1017.000,269.434,-147.954,-25.955,21.420,-31.029
C08762=1016.988,269.678,-148.007,-25.992,21.439,-30.791
C08763=1016.975,269.922,-148.060,-26.030,21.459,-30.551
C08764=1016.960,270.201,-148.122,-26.072,21.483,-30.277
C08765=1016.945,270.479,-148.184,-26.115,21.507,-30.003
C08766=1016.929,270.757,-148.247,-26.158,21.533,-29.728
C08767=1016.913,271.035,-148.311,-26.201,21.560,-29.450
C08768=1016.898,271.279,-148.368,-26.238,21.585,-29.208
C08769=1016.883,271.522,-148.425,-26.276,21.610,-28.964
C08770=1016.868,271.765,-148.482,-26.314,21.637,-28.720
C08771=1016.852,272.007,-148.540,-26.351,21.664,-28.476
C08772=1016.834,272.286,-148.607,-26.395,21.697,-28.194
C08773=1016.815,272.563,-148.675,-26.438,21.731,-27.910
C08774=1016.795,272.842,-148.743,-26.481,21.766,-27.626
C08775=1016.775,273.119,-148.812,-26.525,21.803,-27.342
C08776=1016.758,273.361,-148.872,-26.562,21.835,-27.092
C08777=1016.740,273.603,-148.934,-26.600,21.869,-26.841
C08778=1016.721,273.844,-148.996,-26.638,21.903,-26.590
C08779=1016.702,274.086,-149.058,-26.676,21.940,-26.336
C08780=1016.679,274.365,-149.130,-26.720,21.983,-26.043
C08781=1016.657,274.642,-149.204,-26.763,22.027,-25.750
C08782=1016.634,274.919,-149.277,-26.807,22.073,-25.453
C08783=1016.610,275.197,-149.352,-26.851,22.119,-25.156
C08784=1016.589,275.437,-149.417,-26.889,22.162,-24.896
C08785=1016.568,275.678,-149.483,-26.927,22.204,-24.635
C08786=1016.546,275.918,-149.549,-26.965,22.250,-24.373
C08787=1016.524,276.158,-149.616,-27.003,22.294,-24.111
C08788=1016.498,276.435,-149.694,-27.046,22.349,-23.804
C08789=1016.472,276.713,-149.772,-27.090,22.404,-23.496
C08790=1016.444,276.989,-149.852,-27.134,22.462,-23.186
C08791=1016.417,277.266,-149.932,-27.177,22.521,-22.877
C08792=1016.393,277.506,-150.002,-27.215,22.573,-22.606
C08793=1016.367,277.744,-150.072,-27.252,22.626,-22.334
C08794=1016.342,277.983,-150.143,-27.290,22.681,-22.062
C08795=1016.317,278.221,-150.214,-27.327,22.737,-21.789
C08796=1016.287,278.498,-150.298,-27.370,22.804,-21.469
C08797=1016.256,278.775,-150.382,-27.413,22.873,-21.147
C08798=1016.225,279.051,-150.468,-27.456,22.942,-20.824
C08799=1016.194,279.328,-150.553,-27.498,23.014,-20.499
C08800=1016.166,279.564,-150.627,-27.534,23.078,-20.218
C08801=1016.138,279.802,-150.702,-27.570,23.143,-19.936
C08802=1016.109,280.039,-150.778,-27.606,23.208,-19.653
C08803=1016.081,280.275,-150.854,-27.642,23.276,-19.367
C08804=1016.047,280.551,-150.943,-27.684,23.357,-19.031
C08805=1016.012,280.827,-151.034,-27.725,23.440,-18.691
C08806=1015.977,281.103,-151.124,-27.766,23.526,-18.349
C08807=1015.941,281.379,-151.215,-27.807,23.613,-18.004
C08808=1015.910,281.613,-151.295,-27.842,23.690,-17.706
C08809=1015.879,281.849,-151.375,-27.877,23.768,-17.406
C08810=1015.847,282.083,-151.454,-27.911,23.848,-17.104
C08811=1015.815,282.319,-151.535,-27.945,23.929,-16.801
C08812=1015.775,282.594,-151.631,-27.984,24.027,-16.441
C08813=1015.737,282.869,-151.726,-28.023,24.128,-16.079
C08814=1015.698,283.144,-151.824,-28.062,24.232,-15.713
C08815=1015.657,283.418,-151.922,-28.100,24.338,-15.343
C08816=1015.623,283.651,-152.006,-28.132,24.429,-15.026
C08817=1015.588,283.884,-152.090,-28.164,24.524,-14.708
C08818=1015.552,284.117,-152.175,-28.195,24.619,-14.388
C08819=1015.517,284.348,-152.261,-28.226,24.716,-14.065
C08820=1015.474,284.623,-152.362,-28.261,24.835,-13.680
C08821=1015.429,284.897,-152.465,-28.296,24.955,-13.292
C08822=1015.386,285.171,-152.569,-28.330,25.079,-12.901
C08823=1015.341,285.444,-152.674,-28.364,25.204,-12.507
C08824=1015.303,285.674,-152.763,-28.391,25.314,-12.171
C08825=1015.264,285.905,-152.851,-28.418,25.425,-11.832
C08826=1015.226,286.135,-152.941,-28.444,25.537,-11.492
C08827=1015.186,286.365,-153.032,-28.470,25.652,-11.148
C08828=1015.138,286.638,-153.140,-28.499,25.792,-10.737
C08829=1015.090,286.910,-153.251,-28.527,25.936,-10.320
C08830=1015.041,287.182,-153.360,-28.555,26.082,-9.899
C08831=1014.991,287.455,-153.471,-28.581,26.233,-9.471
C08832=1014.949,287.682,-153.565,-28.602,26.363,-9.109
C08833=1014.907,287.910,-153.659,-28.622,26.495,-8.743
C08834=1014.864,288.138,-153.755,-28.641,26.630,-8.372
C08835=1014.821,288.365,-153.851,-28.659,26.767,-7.999
C08836=1014.767,288.636,-153.966,-28.679,26.937,-7.545
C08837=1014.714,288.907,-154.083,-28.698,27.109,-7.088
C08838=1014.661,289.177,-154.200,-28.715,27.285,-6.624
C08839=1014.606,289.447,-154.318,-28.730,27.467,-6.153
C08840=1014.560,289.672,-154.418,-28.742,27.622,-5.757
C08841=1014.514,289.897,-154.517,-28.752,27.779,-5.357
C08842=1014.467,290.121,-154.618,-28.760,27.939,-4.952
C08843=1014.419,290.345,-154.719,-28.767,28.103,-4.544
C08844=1014.361,290.614,-154.842,-28.773,28.305,-4.046
C08845=1014.303,290.883,-154.966,-28.777,28.511,-3.540
C08846=1014.244,291.151,-155.091,-28.778,28.722,-3.030
C08847=1014.184,291.419,-155.217,-28.777,28.937,-2.514
C08848=1014.134,291.640,-155.321,-28.773,29.120,-2.080
C08849=1014.083,291.861,-155.428,-28.768,29.306,-1.642
C08850=1014.032,292.082,-155.533,-28.760,29.494,-1.200
C08851=1013.980,292.302,-155.641,-28.751,29.686,-0.753
C08852=1013.916,292.570,-155.771,-28.736,29.926,-0.203
C08853=1013.853,292.835,-155.903,-28.717,30.168,0.353
C08854=1013.788,293.101,-156.035,-28.695,30.417,0.916
C08855=1013.722,293.367,-156.169,-28.669,30.673,1.490
C08856=1013.667,293.584,-156.280,-28.645,30.886,1.967
C08857=1013.612,293.801,-156.392,-28.617,31.104,2.450
C08858=1013.557,294.018,-156.504,-28.586,31.327,2.940
C08859=1013.501,294.235,-156.617,-28.552,31.552,3.436
C08860=1013.431,294.498,-156.756,-28.506,31.835,4.050
C08861=1013.362,294.761,-156.896,-28.455,32.123,4.674
C08862=1013.290,295.024,-157.037,-28.398,32.417,5.306
C08863=1013.218,295.285,-157.179,-28.335,32.716,5.947
C08864=1013.159,295.498,-157.296,-28.280,32.966,6.479
C08865=1013.099,295.711,-157.414,-28.220,33.220,7.016
C08866=1013.039,295.924,-157.532,-28.156,33.478,7.560
C08867=1012.979,296.136,-157.652,-28.087,33.740,8.111
C08868=1012.903,296.396,-157.800,-27.996,34.069,8.801
C08869=1012.826,296.655,-157.948,-27.897,34.404,9.500
C08870=1012.749,296.914,-158.098,-27.790,34.746,10.213
C08871=1012.670,297.173,-158.250,-27.675,35.094,10.935
C08872=1012.607,297.381,-158.373,-27.576,35.380,11.529
C08873=1012.542,297.588,-158.497,-27.470,35.670,12.129
C08874=1012.477,297.795,-158.621,-27.359,35.964,12.737
C08875=1012.411,298.002,-158.747,-27.241,36.263,13.354
C08876=1012.329,298.258,-158.904,-27.085,36.640,14.133
C08877=1012.245,298.514,-159.062,-26.918,37.024,14.926
C08878=1012.162,298.768,-159.222,-26.741,37.414,15.733
C08879=1012.076,299.023,-159.383,-26.551,37.810,16.553
C08880=1012.007,299.225,-159.513,-26.391,38.132,17.220
C08881=1011.938,299.427,-159.643,-26.221,38.458,17.898
C08882=1011.868,299.628,-159.774,-26.044,38.787,18.584
C08883=1011.798,299.830,-159.906,-25.858,39.120,19.281
///RCONF 0,0,0,0,0,0,0,0,0,0,0,0,0,0,0,0,0,0,0,0,0,0,0,0
C08884=1011.708,300.081,-160.073,-25.611,39.544,20.170
C08885=1011.617,300.332,-160.240,-25.349,39.974,21.077
C08886=1011.527,300.582,-160.411,-25.071,40.409,21.999
C08887=1011.433,300.831,-160.581,-24.778,40.847,22.938
C08888=1011.360,301.026,-160.717,-24.533,41.199,23.695
C08889=1011.285,301.222,-160.854,-24.278,41.553,24.463
C08890=1011.210,301.418,-160.992,-24.011,41.910,25.243
C08891=1011.135,301.612,-161.131,-23.731,42.271,26.037
C08892=1011.037,301.858,-161.307,-23.359,42.732,27.060
C08893=1010.939,302.103,-161.486,-22.967,43.196,28.105
C08894=1010.841,302.347,-161.666,-22.552,43.665,29.173
C08895=1010.741,302.590,-161.846,-22.115,44.137,30.264
C08896=1010.662,302.779,-161.989,-21.757,44.508,31.133
C08897=1010.582,302.968,-162.132,-21.384,44.880,32.017
C08898=1010.502,303.156,-162.277,-20.997,45.253,32.914
C08899=1010.421,303.344,-162.422,-20.593,45.627,33.826
C08900=1010.316,303.584,-162.609,-20.052,46.107,35.019
C08901=1010.210,303.822,-162.797,-19.485,46.587,36.235
C08902=1010.104,304.060,-162.987,-18.890,47.066,37.479
C08903=1009.996,304.296,-163.178,-18.265,47.545,38.750
C08904=1009.912,304.478,-163.328,-17.761,47.914,39.754
C08905=1009.827,304.660,-163.478,-17.238,48.282,40.774
C08906=1009.741,304.841,-163.629,-16.695,48.650,41.816
C08907=1009.656,305.021,-163.780,-16.133,49.014,42.872
C08908=1009.544,305.253,-163.978,-15.374,49.484,44.273
C08909=1009.429,305.485,-164.177,-14.580,49.949,45.706
C08910=1009.315,305.714,-164.377,-13.751,50.408,47.169
C08911=1009.199,305.943,-164.579,-12.888,50.859,48.662
C08912=1009.110,306.117,-164.733,-12.202,51.199,49.829
C08913=1009.021,306.291,-164.890,-11.496,51.534,51.012
C08914=1008.930,306.464,-165.047,-10.767,51.863,52.216
C08915=1008.838,306.636,-165.205,-10.018,52.186,53.439
C08916=1008.718,306.860,-165.412,-9.002,52.599,55.068
C08917=1008.597,307.083,-165.622,-7.948,53.000,56.733
C08918=1008.474,307.304,-165.831,-6.854,53.388,58.434
C08919=1008.351,307.525,-166.044,-5.724,53.761,60.165
C08920=1008.256,307.690,-166.205,-4.837,54.035,61.506
C08921=1008.162,307.856,-166.367,-3.930,54.299,62.863
C08922=1008.066,308.020,-166.530,-2.999,54.554,64.242
C08923=1007.970,308.184,-166.694,-2.047,54.798,65.640
C08924=1007.842,308.399,-166.911,-0.758,55.103,67.512
C08925=1007.714,308.612,-167.129,0.564,55.388,69.411
C08926=1007.584,308.824,-167.350,1.921,55.651,71.337
C08927=1007.453,309.035,-167.571,3.305,55.891,73.285
C08928=1007.328,309.233,-167.781,4.645,56.098,75.153
C08929=1007.201,309.429,-167.992,6.006,56.283,77.036
C08930=1007.063,309.623,-168.196,7.388,56.445,78.933
C08931=1006.911,309.814,-168.392,8.785,56.584,80.835
C08932=1007.227,309.942,-168.744,9.528,56.648,81.844
C08933=1007.405,309.729,-168.525,7.945,56.504,79.693
C08934=1007.567,309.510,-168.298,6.373,56.328,77.540
C08935=1007.714,309.288,-168.060,4.824,56.124,75.402
C08936=1007.855,309.064,-167.821,3.305,55.891,73.285
C08937=1007.986,308.854,-167.600,1.921,55.651,71.337
C08938=1008.116,308.641,-167.380,0.564,55.388,69.411
C08939=1008.244,308.428,-167.162,-0.758,55.103,67.512
C08940=1008.373,308.213,-166.945,-2.047,54.798,65.640
C08941=1008.469,308.049,-166.781,-2.999,54.554,64.242
C08942=1008.564,307.884,-166.617,-3.930,54.299,62.863
C08943=1008.659,307.719,-166.456,-4.837,54.035,61.506
C08944=1008.753,307.553,-166.295,-5.724,53.761,60.165
C08945=1008.877,307.334,-166.082,-6.854,53.388,58.434
C08946=1008.998,307.112,-165.872,-7.948,53.000,56.733
C08947=1009.120,306.889,-165.663,-9.002,52.599,55.068
C08948=1009.240,306.665,-165.455,-10.018,52.186,53.439
C08949=1009.332,306.493,-165.297,-10.767,51.863,52.216
C08950=1009.422,306.320,-165.141,-11.496,51.534,51.012
C08951=1009.512,306.146,-164.984,-12.202,51.199,49.829
C08952=1009.602,305.972,-164.830,-12.888,50.859,48.662
C08953=1009.717,305.743,-164.628,-13.751,50.408,47.169
C08954=1009.832,305.514,-164.428,-14.580,49.949,45.706
C08955=1009.945,305.282,-164.229,-15.374,49.484,44.273
C08956=1010.058,305.050,-164.031,-16.132,49.015,42.875
C08957=1010.144,304.870,-163.880,-16.695,48.650,41.816
C08958=1010.229,304.689,-163.729,-17.238,48.282,40.774
C08959=1010.313,304.508,-163.578,-17.761,47.914,39.754
C08960=1010.398,304.325,-163.429,-18.265,47.545,38.750
